   // UNICODE_TO_GBK[32326] := 16#8A56;
   // UNICODE_TO_GBK[32327] := 16#D476;
   // UNICODE_TO_GBK[32328] := 16#8A57;
   // UNICODE_TO_GBK[32329] := 16#D477;
   // UNICODE_TO_GBK[32330] := 16#8A58;
   // UNICODE_TO_GBK[32331] := 16#D478;
   // UNICODE_TO_GBK[32332] := 16#8A59;
   // UNICODE_TO_GBK[32333] := 16#D479;
   // UNICODE_TO_GBK[32334] := 16#8A5A;
   // UNICODE_TO_GBK[32335] := 16#D47A;
   // UNICODE_TO_GBK[32336] := 16#8A5B;
   // UNICODE_TO_GBK[32337] := 16#D47B;
   // UNICODE_TO_GBK[32338] := 16#8A5C;
   // UNICODE_TO_GBK[32339] := 16#D47C;
   // UNICODE_TO_GBK[32340] := 16#8A5D;
   // UNICODE_TO_GBK[32341] := 16#D47D;
   // UNICODE_TO_GBK[32342] := 16#8A5E;
   // UNICODE_TO_GBK[32343] := 16#D47E;
   // UNICODE_TO_GBK[32344] := 16#8A5F;
   // UNICODE_TO_GBK[32345] := 16#D480;
   // UNICODE_TO_GBK[32346] := 16#8A60;
   // UNICODE_TO_GBK[32347] := 16#D481;
   // UNICODE_TO_GBK[32348] := 16#8A61;
   // UNICODE_TO_GBK[32349] := 16#D482;
   // UNICODE_TO_GBK[32350] := 16#8A62;
   // UNICODE_TO_GBK[32351] := 16#D483;
   // UNICODE_TO_GBK[32352] := 16#8A63;
   // UNICODE_TO_GBK[32353] := 16#D484;
   // UNICODE_TO_GBK[32354] := 16#8A64;
   // UNICODE_TO_GBK[32355] := 16#D485;
   // UNICODE_TO_GBK[32356] := 16#8A65;
   // UNICODE_TO_GBK[32357] := 16#D486;
   // UNICODE_TO_GBK[32358] := 16#8A66;
   // UNICODE_TO_GBK[32359] := 16#D487;
   // UNICODE_TO_GBK[32360] := 16#8A67;
   // UNICODE_TO_GBK[32361] := 16#D488;
   // UNICODE_TO_GBK[32362] := 16#8A68;
   // UNICODE_TO_GBK[32363] := 16#D489;
   // UNICODE_TO_GBK[32364] := 16#8A69;
   // UNICODE_TO_GBK[32365] := 16#D48A;
   // UNICODE_TO_GBK[32366] := 16#8A6A;
   // UNICODE_TO_GBK[32367] := 16#D48B;
   // UNICODE_TO_GBK[32368] := 16#8A6B;
   // UNICODE_TO_GBK[32369] := 16#D48C;
   // UNICODE_TO_GBK[32370] := 16#8A6C;
   // UNICODE_TO_GBK[32371] := 16#D48D;
   // UNICODE_TO_GBK[32372] := 16#8A6D;
   // UNICODE_TO_GBK[32373] := 16#D48E;
   // UNICODE_TO_GBK[32374] := 16#8A6E;
   // UNICODE_TO_GBK[32375] := 16#D48F;
   // UNICODE_TO_GBK[32376] := 16#8A6F;
   // UNICODE_TO_GBK[32377] := 16#D490;
   // UNICODE_TO_GBK[32378] := 16#8A70;
   // UNICODE_TO_GBK[32379] := 16#D491;
   // UNICODE_TO_GBK[32380] := 16#8A71;
   // UNICODE_TO_GBK[32381] := 16#D492;
   // UNICODE_TO_GBK[32382] := 16#8A72;
   // UNICODE_TO_GBK[32383] := 16#D493;
   // UNICODE_TO_GBK[32384] := 16#8A73;
   // UNICODE_TO_GBK[32385] := 16#D494;
   // UNICODE_TO_GBK[32386] := 16#8A74;
   // UNICODE_TO_GBK[32387] := 16#D495;
   // UNICODE_TO_GBK[32388] := 16#8A75;
   // UNICODE_TO_GBK[32389] := 16#D496;
   // UNICODE_TO_GBK[32390] := 16#8A76;
   // UNICODE_TO_GBK[32391] := 16#D497;
   // UNICODE_TO_GBK[32392] := 16#8A77;
   // UNICODE_TO_GBK[32393] := 16#D498;
   // UNICODE_TO_GBK[32394] := 16#8A78;
   // UNICODE_TO_GBK[32395] := 16#D499;
   // UNICODE_TO_GBK[32396] := 16#8A79;
   // UNICODE_TO_GBK[32397] := 16#D5B2;
   // UNICODE_TO_GBK[32398] := 16#8A7A;
   // UNICODE_TO_GBK[32399] := 16#D49A;
   // UNICODE_TO_GBK[32400] := 16#8A7B;
   // UNICODE_TO_GBK[32401] := 16#D49B;
   // UNICODE_TO_GBK[32402] := 16#8A7C;
   // UNICODE_TO_GBK[32403] := 16#D49C;
   // UNICODE_TO_GBK[32404] := 16#8A7D;
   // UNICODE_TO_GBK[32405] := 16#D49D;
   // UNICODE_TO_GBK[32406] := 16#8A7E;
   // UNICODE_TO_GBK[32407] := 16#D49E;
   // UNICODE_TO_GBK[32408] := 16#8A7F;
   // UNICODE_TO_GBK[32409] := 16#D49F;
   // UNICODE_TO_GBK[32410] := 16#8A80;
   // UNICODE_TO_GBK[32411] := 16#D4A0;
   // UNICODE_TO_GBK[32412] := 16#8A81;
   // UNICODE_TO_GBK[32413] := 16#D540;
   // UNICODE_TO_GBK[32414] := 16#8A82;
   // UNICODE_TO_GBK[32415] := 16#D541;
   // UNICODE_TO_GBK[32416] := 16#8A83;
   // UNICODE_TO_GBK[32417] := 16#D542;
   // UNICODE_TO_GBK[32418] := 16#8A84;
   // UNICODE_TO_GBK[32419] := 16#D543;
   // UNICODE_TO_GBK[32420] := 16#8A85;
   // UNICODE_TO_GBK[32421] := 16#D544;
   // UNICODE_TO_GBK[32422] := 16#8A86;
   // UNICODE_TO_GBK[32423] := 16#D545;
   // UNICODE_TO_GBK[32424] := 16#8A87;
   // UNICODE_TO_GBK[32425] := 16#D546;
   // UNICODE_TO_GBK[32426] := 16#8A88;
   // UNICODE_TO_GBK[32427] := 16#D547;
   // UNICODE_TO_GBK[32428] := 16#8A89;
   // UNICODE_TO_GBK[32429] := 16#D3FE;
   // UNICODE_TO_GBK[32430] := 16#8A8A;
   // UNICODE_TO_GBK[32431] := 16#CCDC;
   // UNICODE_TO_GBK[32432] := 16#8A8B;
   // UNICODE_TO_GBK[32433] := 16#D548;
   // UNICODE_TO_GBK[32434] := 16#8A8C;
   // UNICODE_TO_GBK[32435] := 16#D549;
   // UNICODE_TO_GBK[32436] := 16#8A8D;
   // UNICODE_TO_GBK[32437] := 16#D54A;
   // UNICODE_TO_GBK[32438] := 16#8A8E;
   // UNICODE_TO_GBK[32439] := 16#D54B;
   // UNICODE_TO_GBK[32440] := 16#8A8F;
   // UNICODE_TO_GBK[32441] := 16#D54C;
   // UNICODE_TO_GBK[32442] := 16#8A90;
   // UNICODE_TO_GBK[32443] := 16#D54D;
   // UNICODE_TO_GBK[32444] := 16#8A91;
   // UNICODE_TO_GBK[32445] := 16#D54E;
   // UNICODE_TO_GBK[32446] := 16#8A92;
   // UNICODE_TO_GBK[32447] := 16#D54F;
   // UNICODE_TO_GBK[32448] := 16#8A93;
   // UNICODE_TO_GBK[32449] := 16#CAC4;
   // UNICODE_TO_GBK[32450] := 16#8A94;
   // UNICODE_TO_GBK[32451] := 16#D550;
   // UNICODE_TO_GBK[32452] := 16#8A95;
   // UNICODE_TO_GBK[32453] := 16#D551;
   // UNICODE_TO_GBK[32454] := 16#8A96;
   // UNICODE_TO_GBK[32455] := 16#D552;
   // UNICODE_TO_GBK[32456] := 16#8A97;
   // UNICODE_TO_GBK[32457] := 16#D553;
   // UNICODE_TO_GBK[32458] := 16#8A98;
   // UNICODE_TO_GBK[32459] := 16#D554;
   // UNICODE_TO_GBK[32460] := 16#8A99;
   // UNICODE_TO_GBK[32461] := 16#D555;
   // UNICODE_TO_GBK[32462] := 16#8A9A;
   // UNICODE_TO_GBK[32463] := 16#D556;
   // UNICODE_TO_GBK[32464] := 16#8A9B;
   // UNICODE_TO_GBK[32465] := 16#D557;
   // UNICODE_TO_GBK[32466] := 16#8A9C;
   // UNICODE_TO_GBK[32467] := 16#D558;
   // UNICODE_TO_GBK[32468] := 16#8A9D;
   // UNICODE_TO_GBK[32469] := 16#D559;
   // UNICODE_TO_GBK[32470] := 16#8A9E;
   // UNICODE_TO_GBK[32471] := 16#D55A;
   // UNICODE_TO_GBK[32472] := 16#8A9F;
   // UNICODE_TO_GBK[32473] := 16#D55B;
   // UNICODE_TO_GBK[32474] := 16#8AA0;
   // UNICODE_TO_GBK[32475] := 16#D55C;
   // UNICODE_TO_GBK[32476] := 16#8AA1;
   // UNICODE_TO_GBK[32477] := 16#D55D;
   // UNICODE_TO_GBK[32478] := 16#8AA2;
   // UNICODE_TO_GBK[32479] := 16#D55E;
   // UNICODE_TO_GBK[32480] := 16#8AA3;
   // UNICODE_TO_GBK[32481] := 16#D55F;
   // UNICODE_TO_GBK[32482] := 16#8AA4;
   // UNICODE_TO_GBK[32483] := 16#D560;
   // UNICODE_TO_GBK[32484] := 16#8AA5;
   // UNICODE_TO_GBK[32485] := 16#D561;
   // UNICODE_TO_GBK[32486] := 16#8AA6;
   // UNICODE_TO_GBK[32487] := 16#D562;
   // UNICODE_TO_GBK[32488] := 16#8AA7;
   // UNICODE_TO_GBK[32489] := 16#D563;
   // UNICODE_TO_GBK[32490] := 16#8AA8;
   // UNICODE_TO_GBK[32491] := 16#D564;
   // UNICODE_TO_GBK[32492] := 16#8AA9;
   // UNICODE_TO_GBK[32493] := 16#D565;
   // UNICODE_TO_GBK[32494] := 16#8AAA;
   // UNICODE_TO_GBK[32495] := 16#D566;
   // UNICODE_TO_GBK[32496] := 16#8AAB;
   // UNICODE_TO_GBK[32497] := 16#D567;
   // UNICODE_TO_GBK[32498] := 16#8AAC;
   // UNICODE_TO_GBK[32499] := 16#D568;
   // UNICODE_TO_GBK[32500] := 16#8AAD;
   // UNICODE_TO_GBK[32501] := 16#D569;
   // UNICODE_TO_GBK[32502] := 16#8AAE;
   // UNICODE_TO_GBK[32503] := 16#D56A;
   // UNICODE_TO_GBK[32504] := 16#8AAF;
   // UNICODE_TO_GBK[32505] := 16#D56B;
   // UNICODE_TO_GBK[32506] := 16#8AB0;
   // UNICODE_TO_GBK[32507] := 16#D56C;
   // UNICODE_TO_GBK[32508] := 16#8AB1;
   // UNICODE_TO_GBK[32509] := 16#D56D;
   // UNICODE_TO_GBK[32510] := 16#8AB2;
   // UNICODE_TO_GBK[32511] := 16#D56E;
   // UNICODE_TO_GBK[32512] := 16#8AB3;
   // UNICODE_TO_GBK[32513] := 16#D56F;
   // UNICODE_TO_GBK[32514] := 16#8AB4;
   // UNICODE_TO_GBK[32515] := 16#D570;
   // UNICODE_TO_GBK[32516] := 16#8AB5;
   // UNICODE_TO_GBK[32517] := 16#D571;
   // UNICODE_TO_GBK[32518] := 16#8AB6;
   // UNICODE_TO_GBK[32519] := 16#D572;
   // UNICODE_TO_GBK[32520] := 16#8AB7;
   // UNICODE_TO_GBK[32521] := 16#D573;
   // UNICODE_TO_GBK[32522] := 16#8AB8;
   // UNICODE_TO_GBK[32523] := 16#D574;
   // UNICODE_TO_GBK[32524] := 16#8AB9;
   // UNICODE_TO_GBK[32525] := 16#D575;
   // UNICODE_TO_GBK[32526] := 16#8ABA;
   // UNICODE_TO_GBK[32527] := 16#D576;
   // UNICODE_TO_GBK[32528] := 16#8ABB;
   // UNICODE_TO_GBK[32529] := 16#D577;
   // UNICODE_TO_GBK[32530] := 16#8ABC;
   // UNICODE_TO_GBK[32531] := 16#D578;
   // UNICODE_TO_GBK[32532] := 16#8ABD;
   // UNICODE_TO_GBK[32533] := 16#D579;
   // UNICODE_TO_GBK[32534] := 16#8ABE;
   // UNICODE_TO_GBK[32535] := 16#D57A;
   // UNICODE_TO_GBK[32536] := 16#8ABF;
   // UNICODE_TO_GBK[32537] := 16#D57B;
   // UNICODE_TO_GBK[32538] := 16#8AC0;
   // UNICODE_TO_GBK[32539] := 16#D57C;
   // UNICODE_TO_GBK[32540] := 16#8AC1;
   // UNICODE_TO_GBK[32541] := 16#D57D;
   // UNICODE_TO_GBK[32542] := 16#8AC2;
   // UNICODE_TO_GBK[32543] := 16#D57E;
   // UNICODE_TO_GBK[32544] := 16#8AC3;
   // UNICODE_TO_GBK[32545] := 16#D580;
   // UNICODE_TO_GBK[32546] := 16#8AC4;
   // UNICODE_TO_GBK[32547] := 16#D581;
   // UNICODE_TO_GBK[32548] := 16#8AC5;
   // UNICODE_TO_GBK[32549] := 16#D582;
   // UNICODE_TO_GBK[32550] := 16#8AC6;
   // UNICODE_TO_GBK[32551] := 16#D583;
   // UNICODE_TO_GBK[32552] := 16#8AC7;
   // UNICODE_TO_GBK[32553] := 16#D584;
   // UNICODE_TO_GBK[32554] := 16#8AC8;
   // UNICODE_TO_GBK[32555] := 16#D585;
   // UNICODE_TO_GBK[32556] := 16#8AC9;
   // UNICODE_TO_GBK[32557] := 16#D586;
   // UNICODE_TO_GBK[32558] := 16#8ACA;
   // UNICODE_TO_GBK[32559] := 16#D587;
   // UNICODE_TO_GBK[32560] := 16#8ACB;
   // UNICODE_TO_GBK[32561] := 16#D588;
   // UNICODE_TO_GBK[32562] := 16#8ACC;
   // UNICODE_TO_GBK[32563] := 16#D589;
   // UNICODE_TO_GBK[32564] := 16#8ACD;
   // UNICODE_TO_GBK[32565] := 16#D58A;
   // UNICODE_TO_GBK[32566] := 16#8ACE;
   // UNICODE_TO_GBK[32567] := 16#D58B;
   // UNICODE_TO_GBK[32568] := 16#8ACF;
   // UNICODE_TO_GBK[32569] := 16#D58C;
   // UNICODE_TO_GBK[32570] := 16#8AD0;
   // UNICODE_TO_GBK[32571] := 16#D58D;
   // UNICODE_TO_GBK[32572] := 16#8AD1;
   // UNICODE_TO_GBK[32573] := 16#D58E;
   // UNICODE_TO_GBK[32574] := 16#8AD2;
   // UNICODE_TO_GBK[32575] := 16#D58F;
   // UNICODE_TO_GBK[32576] := 16#8AD3;
   // UNICODE_TO_GBK[32577] := 16#D590;
   // UNICODE_TO_GBK[32578] := 16#8AD4;
   // UNICODE_TO_GBK[32579] := 16#D591;
   // UNICODE_TO_GBK[32580] := 16#8AD5;
   // UNICODE_TO_GBK[32581] := 16#D592;
   // UNICODE_TO_GBK[32582] := 16#8AD6;
   // UNICODE_TO_GBK[32583] := 16#D593;
   // UNICODE_TO_GBK[32584] := 16#8AD7;
   // UNICODE_TO_GBK[32585] := 16#D594;
   // UNICODE_TO_GBK[32586] := 16#8AD8;
   // UNICODE_TO_GBK[32587] := 16#D595;
   // UNICODE_TO_GBK[32588] := 16#8AD9;
   // UNICODE_TO_GBK[32589] := 16#D596;
   // UNICODE_TO_GBK[32590] := 16#8ADA;
   // UNICODE_TO_GBK[32591] := 16#D597;
   // UNICODE_TO_GBK[32592] := 16#8ADB;
   // UNICODE_TO_GBK[32593] := 16#D598;
   // UNICODE_TO_GBK[32594] := 16#8ADC;
   // UNICODE_TO_GBK[32595] := 16#D599;
   // UNICODE_TO_GBK[32596] := 16#8ADD;
   // UNICODE_TO_GBK[32597] := 16#D59A;
   // UNICODE_TO_GBK[32598] := 16#8ADE;
   // UNICODE_TO_GBK[32599] := 16#D59B;
   // UNICODE_TO_GBK[32600] := 16#8ADF;
   // UNICODE_TO_GBK[32601] := 16#D59C;
   // UNICODE_TO_GBK[32602] := 16#8AE0;
   // UNICODE_TO_GBK[32603] := 16#D59D;
   // UNICODE_TO_GBK[32604] := 16#8AE1;
   // UNICODE_TO_GBK[32605] := 16#D59E;
   // UNICODE_TO_GBK[32606] := 16#8AE2;
   // UNICODE_TO_GBK[32607] := 16#D59F;
   // UNICODE_TO_GBK[32608] := 16#8AE3;
   // UNICODE_TO_GBK[32609] := 16#D5A0;
   // UNICODE_TO_GBK[32610] := 16#8AE4;
   // UNICODE_TO_GBK[32611] := 16#D640;
   // UNICODE_TO_GBK[32612] := 16#8AE5;
   // UNICODE_TO_GBK[32613] := 16#D641;
   // UNICODE_TO_GBK[32614] := 16#8AE6;
   // UNICODE_TO_GBK[32615] := 16#D642;
   // UNICODE_TO_GBK[32616] := 16#8AE7;
   // UNICODE_TO_GBK[32617] := 16#D643;
   // UNICODE_TO_GBK[32618] := 16#8AE8;
   // UNICODE_TO_GBK[32619] := 16#D644;
   // UNICODE_TO_GBK[32620] := 16#8AE9;
   // UNICODE_TO_GBK[32621] := 16#D645;
   // UNICODE_TO_GBK[32622] := 16#8AEA;
   // UNICODE_TO_GBK[32623] := 16#D646;
   // UNICODE_TO_GBK[32624] := 16#8AEB;
   // UNICODE_TO_GBK[32625] := 16#D647;
   // UNICODE_TO_GBK[32626] := 16#8AEC;
   // UNICODE_TO_GBK[32627] := 16#D648;
   // UNICODE_TO_GBK[32628] := 16#8AED;
   // UNICODE_TO_GBK[32629] := 16#D649;
   // UNICODE_TO_GBK[32630] := 16#8AEE;
   // UNICODE_TO_GBK[32631] := 16#D64A;
   // UNICODE_TO_GBK[32632] := 16#8AEF;
   // UNICODE_TO_GBK[32633] := 16#D64B;
   // UNICODE_TO_GBK[32634] := 16#8AF0;
   // UNICODE_TO_GBK[32635] := 16#D64C;
   // UNICODE_TO_GBK[32636] := 16#8AF1;
   // UNICODE_TO_GBK[32637] := 16#D64D;
   // UNICODE_TO_GBK[32638] := 16#8AF2;
   // UNICODE_TO_GBK[32639] := 16#D64E;
   // UNICODE_TO_GBK[32640] := 16#8AF3;
   // UNICODE_TO_GBK[32641] := 16#D64F;
   // UNICODE_TO_GBK[32642] := 16#8AF4;
   // UNICODE_TO_GBK[32643] := 16#D650;
   // UNICODE_TO_GBK[32644] := 16#8AF5;
   // UNICODE_TO_GBK[32645] := 16#D651;
   // UNICODE_TO_GBK[32646] := 16#8AF6;
   // UNICODE_TO_GBK[32647] := 16#D652;
   // UNICODE_TO_GBK[32648] := 16#8AF7;
   // UNICODE_TO_GBK[32649] := 16#D653;
   // UNICODE_TO_GBK[32650] := 16#8AF8;
   // UNICODE_TO_GBK[32651] := 16#D654;
   // UNICODE_TO_GBK[32652] := 16#8AF9;
   // UNICODE_TO_GBK[32653] := 16#D655;
   // UNICODE_TO_GBK[32654] := 16#8AFA;
   // UNICODE_TO_GBK[32655] := 16#D656;
   // UNICODE_TO_GBK[32656] := 16#8AFB;
   // UNICODE_TO_GBK[32657] := 16#D657;
   // UNICODE_TO_GBK[32658] := 16#8AFC;
   // UNICODE_TO_GBK[32659] := 16#D658;
   // UNICODE_TO_GBK[32660] := 16#8AFD;
   // UNICODE_TO_GBK[32661] := 16#D659;
   // UNICODE_TO_GBK[32662] := 16#8AFE;
   // UNICODE_TO_GBK[32663] := 16#D65A;
   // UNICODE_TO_GBK[32664] := 16#8AFF;
   // UNICODE_TO_GBK[32665] := 16#D65B;
   // UNICODE_TO_GBK[32666] := 16#8B00;
   // UNICODE_TO_GBK[32667] := 16#D65C;
   // UNICODE_TO_GBK[32668] := 16#8B01;
   // UNICODE_TO_GBK[32669] := 16#D65D;
   // UNICODE_TO_GBK[32670] := 16#8B02;
   // UNICODE_TO_GBK[32671] := 16#D65E;
   // UNICODE_TO_GBK[32672] := 16#8B03;
   // UNICODE_TO_GBK[32673] := 16#D65F;
   // UNICODE_TO_GBK[32674] := 16#8B04;
   // UNICODE_TO_GBK[32675] := 16#D660;
   // UNICODE_TO_GBK[32676] := 16#8B05;
   // UNICODE_TO_GBK[32677] := 16#D661;
   // UNICODE_TO_GBK[32678] := 16#8B06;
   // UNICODE_TO_GBK[32679] := 16#D662;
   // UNICODE_TO_GBK[32680] := 16#8B07;
   // UNICODE_TO_GBK[32681] := 16#E5C0;
   // UNICODE_TO_GBK[32682] := 16#8B08;
   // UNICODE_TO_GBK[32683] := 16#D663;
   // UNICODE_TO_GBK[32684] := 16#8B09;
   // UNICODE_TO_GBK[32685] := 16#D664;
   // UNICODE_TO_GBK[32686] := 16#8B0A;
   // UNICODE_TO_GBK[32687] := 16#D665;
   // UNICODE_TO_GBK[32688] := 16#8B0B;
   // UNICODE_TO_GBK[32689] := 16#D666;
   // UNICODE_TO_GBK[32690] := 16#8B0C;
   // UNICODE_TO_GBK[32691] := 16#D667;
   // UNICODE_TO_GBK[32692] := 16#8B0D;
   // UNICODE_TO_GBK[32693] := 16#D668;
   // UNICODE_TO_GBK[32694] := 16#8B0E;
   // UNICODE_TO_GBK[32695] := 16#D669;
   // UNICODE_TO_GBK[32696] := 16#8B0F;
   // UNICODE_TO_GBK[32697] := 16#D66A;
   // UNICODE_TO_GBK[32698] := 16#8B10;
   // UNICODE_TO_GBK[32699] := 16#D66B;
   // UNICODE_TO_GBK[32700] := 16#8B11;
   // UNICODE_TO_GBK[32701] := 16#D66C;
   // UNICODE_TO_GBK[32702] := 16#8B12;
   // UNICODE_TO_GBK[32703] := 16#D66D;
   // UNICODE_TO_GBK[32704] := 16#8B13;
   // UNICODE_TO_GBK[32705] := 16#D66E;
   // UNICODE_TO_GBK[32706] := 16#8B14;
   // UNICODE_TO_GBK[32707] := 16#D66F;
   // UNICODE_TO_GBK[32708] := 16#8B15;
   // UNICODE_TO_GBK[32709] := 16#D670;
   // UNICODE_TO_GBK[32710] := 16#8B16;
   // UNICODE_TO_GBK[32711] := 16#D671;
   // UNICODE_TO_GBK[32712] := 16#8B17;
   // UNICODE_TO_GBK[32713] := 16#D672;
   // UNICODE_TO_GBK[32714] := 16#8B18;
   // UNICODE_TO_GBK[32715] := 16#D673;
   // UNICODE_TO_GBK[32716] := 16#8B19;
   // UNICODE_TO_GBK[32717] := 16#D674;
   // UNICODE_TO_GBK[32718] := 16#8B1A;
   // UNICODE_TO_GBK[32719] := 16#D675;
   // UNICODE_TO_GBK[32720] := 16#8B1B;
   // UNICODE_TO_GBK[32721] := 16#D676;
   // UNICODE_TO_GBK[32722] := 16#8B1C;
   // UNICODE_TO_GBK[32723] := 16#D677;
   // UNICODE_TO_GBK[32724] := 16#8B1D;
   // UNICODE_TO_GBK[32725] := 16#D678;
   // UNICODE_TO_GBK[32726] := 16#8B1E;
   // UNICODE_TO_GBK[32727] := 16#D679;
   // UNICODE_TO_GBK[32728] := 16#8B1F;
   // UNICODE_TO_GBK[32729] := 16#D67A;
   // UNICODE_TO_GBK[32730] := 16#8B20;
   // UNICODE_TO_GBK[32731] := 16#D67B;
   // UNICODE_TO_GBK[32732] := 16#8B21;
   // UNICODE_TO_GBK[32733] := 16#D67C;
   // UNICODE_TO_GBK[32734] := 16#8B22;
   // UNICODE_TO_GBK[32735] := 16#D67D;
   // UNICODE_TO_GBK[32736] := 16#8B23;
   // UNICODE_TO_GBK[32737] := 16#D67E;
   // UNICODE_TO_GBK[32738] := 16#8B24;
   // UNICODE_TO_GBK[32739] := 16#D680;
   // UNICODE_TO_GBK[32740] := 16#8B25;
   // UNICODE_TO_GBK[32741] := 16#D681;
   // UNICODE_TO_GBK[32742] := 16#8B26;
   // UNICODE_TO_GBK[32743] := 16#F6A5;
   // UNICODE_TO_GBK[32744] := 16#8B27;
   // UNICODE_TO_GBK[32745] := 16#D682;
   // UNICODE_TO_GBK[32746] := 16#8B28;
   // UNICODE_TO_GBK[32747] := 16#D683;
   // UNICODE_TO_GBK[32748] := 16#8B29;
   // UNICODE_TO_GBK[32749] := 16#D684;
   // UNICODE_TO_GBK[32750] := 16#8B2A;
   // UNICODE_TO_GBK[32751] := 16#D685;
   // UNICODE_TO_GBK[32752] := 16#8B2B;
   // UNICODE_TO_GBK[32753] := 16#D686;
   // UNICODE_TO_GBK[32754] := 16#8B2C;
   // UNICODE_TO_GBK[32755] := 16#D687;
   // UNICODE_TO_GBK[32756] := 16#8B2D;
   // UNICODE_TO_GBK[32757] := 16#D688;
   // UNICODE_TO_GBK[32758] := 16#8B2E;
   // UNICODE_TO_GBK[32759] := 16#D689;
   // UNICODE_TO_GBK[32760] := 16#8B2F;
   // UNICODE_TO_GBK[32761] := 16#D68A;
   // UNICODE_TO_GBK[32762] := 16#8B30;
   // UNICODE_TO_GBK[32763] := 16#D68B;
   // UNICODE_TO_GBK[32764] := 16#8B31;
   // UNICODE_TO_GBK[32765] := 16#D68C;
   // UNICODE_TO_GBK[32766] := 16#8B32;
   // UNICODE_TO_GBK[32767] := 16#D68D;
   // UNICODE_TO_GBK[32768] := 16#8B33;
   // UNICODE_TO_GBK[32769] := 16#D68E;
   // UNICODE_TO_GBK[32770] := 16#8B34;
   // UNICODE_TO_GBK[32771] := 16#D68F;
   // UNICODE_TO_GBK[32772] := 16#8B35;
   // UNICODE_TO_GBK[32773] := 16#D690;
   // UNICODE_TO_GBK[32774] := 16#8B36;
   // UNICODE_TO_GBK[32775] := 16#D691;
   // UNICODE_TO_GBK[32776] := 16#8B37;
   // UNICODE_TO_GBK[32777] := 16#D692;
   // UNICODE_TO_GBK[32778] := 16#8B38;
   // UNICODE_TO_GBK[32779] := 16#D693;
   // UNICODE_TO_GBK[32780] := 16#8B39;
   // UNICODE_TO_GBK[32781] := 16#D694;
   // UNICODE_TO_GBK[32782] := 16#8B3A;
   // UNICODE_TO_GBK[32783] := 16#D695;
   // UNICODE_TO_GBK[32784] := 16#8B3B;
   // UNICODE_TO_GBK[32785] := 16#D696;
   // UNICODE_TO_GBK[32786] := 16#8B3C;
   // UNICODE_TO_GBK[32787] := 16#D697;
   // UNICODE_TO_GBK[32788] := 16#8B3D;
   // UNICODE_TO_GBK[32789] := 16#D698;
   // UNICODE_TO_GBK[32790] := 16#8B3E;
   // UNICODE_TO_GBK[32791] := 16#D699;
   // UNICODE_TO_GBK[32792] := 16#8B3F;
   // UNICODE_TO_GBK[32793] := 16#D69A;
   // UNICODE_TO_GBK[32794] := 16#8B40;
   // UNICODE_TO_GBK[32795] := 16#D69B;
   // UNICODE_TO_GBK[32796] := 16#8B41;
   // UNICODE_TO_GBK[32797] := 16#D69C;
   // UNICODE_TO_GBK[32798] := 16#8B42;
   // UNICODE_TO_GBK[32799] := 16#D69D;
   // UNICODE_TO_GBK[32800] := 16#8B43;
   // UNICODE_TO_GBK[32801] := 16#D69E;
   // UNICODE_TO_GBK[32802] := 16#8B44;
   // UNICODE_TO_GBK[32803] := 16#D69F;
   // UNICODE_TO_GBK[32804] := 16#8B45;
   // UNICODE_TO_GBK[32805] := 16#D6A0;
   // UNICODE_TO_GBK[32806] := 16#8B46;
   // UNICODE_TO_GBK[32807] := 16#D740;
   // UNICODE_TO_GBK[32808] := 16#8B47;
   // UNICODE_TO_GBK[32809] := 16#D741;
   // UNICODE_TO_GBK[32810] := 16#8B48;
   // UNICODE_TO_GBK[32811] := 16#D742;
   // UNICODE_TO_GBK[32812] := 16#8B49;
   // UNICODE_TO_GBK[32813] := 16#D743;
   // UNICODE_TO_GBK[32814] := 16#8B4A;
   // UNICODE_TO_GBK[32815] := 16#D744;
   // UNICODE_TO_GBK[32816] := 16#8B4B;
   // UNICODE_TO_GBK[32817] := 16#D745;
   // UNICODE_TO_GBK[32818] := 16#8B4C;
   // UNICODE_TO_GBK[32819] := 16#D746;
   // UNICODE_TO_GBK[32820] := 16#8B4D;
   // UNICODE_TO_GBK[32821] := 16#D747;
   // UNICODE_TO_GBK[32822] := 16#8B4E;
   // UNICODE_TO_GBK[32823] := 16#D748;
   // UNICODE_TO_GBK[32824] := 16#8B4F;
   // UNICODE_TO_GBK[32825] := 16#D749;
   // UNICODE_TO_GBK[32826] := 16#8B50;
   // UNICODE_TO_GBK[32827] := 16#D74A;
   // UNICODE_TO_GBK[32828] := 16#8B51;
   // UNICODE_TO_GBK[32829] := 16#D74B;
   // UNICODE_TO_GBK[32830] := 16#8B52;
   // UNICODE_TO_GBK[32831] := 16#D74C;
   // UNICODE_TO_GBK[32832] := 16#8B53;
   // UNICODE_TO_GBK[32833] := 16#D74D;
   // UNICODE_TO_GBK[32834] := 16#8B54;
   // UNICODE_TO_GBK[32835] := 16#D74E;
   // UNICODE_TO_GBK[32836] := 16#8B55;
   // UNICODE_TO_GBK[32837] := 16#D74F;
   // UNICODE_TO_GBK[32838] := 16#8B56;
   // UNICODE_TO_GBK[32839] := 16#D750;
   // UNICODE_TO_GBK[32840] := 16#8B57;
   // UNICODE_TO_GBK[32841] := 16#D751;
   // UNICODE_TO_GBK[32842] := 16#8B58;
   // UNICODE_TO_GBK[32843] := 16#D752;
   // UNICODE_TO_GBK[32844] := 16#8B59;
   // UNICODE_TO_GBK[32845] := 16#D753;
   // UNICODE_TO_GBK[32846] := 16#8B5A;
   // UNICODE_TO_GBK[32847] := 16#D754;
   // UNICODE_TO_GBK[32848] := 16#8B5B;
   // UNICODE_TO_GBK[32849] := 16#D755;
   // UNICODE_TO_GBK[32850] := 16#8B5C;
   // UNICODE_TO_GBK[32851] := 16#D756;
   // UNICODE_TO_GBK[32852] := 16#8B5D;
   // UNICODE_TO_GBK[32853] := 16#D757;
   // UNICODE_TO_GBK[32854] := 16#8B5E;
   // UNICODE_TO_GBK[32855] := 16#D758;
   // UNICODE_TO_GBK[32856] := 16#8B5F;
   // UNICODE_TO_GBK[32857] := 16#D759;
   // UNICODE_TO_GBK[32858] := 16#8B60;
   // UNICODE_TO_GBK[32859] := 16#D75A;
   // UNICODE_TO_GBK[32860] := 16#8B61;
   // UNICODE_TO_GBK[32861] := 16#D75B;
   // UNICODE_TO_GBK[32862] := 16#8B62;
   // UNICODE_TO_GBK[32863] := 16#D75C;
   // UNICODE_TO_GBK[32864] := 16#8B63;
   // UNICODE_TO_GBK[32865] := 16#D75D;
   // UNICODE_TO_GBK[32866] := 16#8B64;
   // UNICODE_TO_GBK[32867] := 16#D75E;
   // UNICODE_TO_GBK[32868] := 16#8B65;
   // UNICODE_TO_GBK[32869] := 16#D75F;
   // UNICODE_TO_GBK[32870] := 16#8B66;
   // UNICODE_TO_GBK[32871] := 16#BEAF;
   // UNICODE_TO_GBK[32872] := 16#8B67;
   // UNICODE_TO_GBK[32873] := 16#D760;
   // UNICODE_TO_GBK[32874] := 16#8B68;
   // UNICODE_TO_GBK[32875] := 16#D761;
   // UNICODE_TO_GBK[32876] := 16#8B69;
   // UNICODE_TO_GBK[32877] := 16#D762;
   // UNICODE_TO_GBK[32878] := 16#8B6A;
   // UNICODE_TO_GBK[32879] := 16#D763;
   // UNICODE_TO_GBK[32880] := 16#8B6B;
   // UNICODE_TO_GBK[32881] := 16#D764;
   // UNICODE_TO_GBK[32882] := 16#8B6C;
   // UNICODE_TO_GBK[32883] := 16#C6A9;
   // UNICODE_TO_GBK[32884] := 16#8B6D;
   // UNICODE_TO_GBK[32885] := 16#D765;
   // UNICODE_TO_GBK[32886] := 16#8B6E;
   // UNICODE_TO_GBK[32887] := 16#D766;
   // UNICODE_TO_GBK[32888] := 16#8B6F;
   // UNICODE_TO_GBK[32889] := 16#D767;
   // UNICODE_TO_GBK[32890] := 16#8B70;
   // UNICODE_TO_GBK[32891] := 16#D768;
   // UNICODE_TO_GBK[32892] := 16#8B71;
   // UNICODE_TO_GBK[32893] := 16#D769;
   // UNICODE_TO_GBK[32894] := 16#8B72;
   // UNICODE_TO_GBK[32895] := 16#D76A;
   // UNICODE_TO_GBK[32896] := 16#8B73;
   // UNICODE_TO_GBK[32897] := 16#D76B;
   // UNICODE_TO_GBK[32898] := 16#8B74;
   // UNICODE_TO_GBK[32899] := 16#D76C;
   // UNICODE_TO_GBK[32900] := 16#8B75;
   // UNICODE_TO_GBK[32901] := 16#D76D;
   // UNICODE_TO_GBK[32902] := 16#8B76;
   // UNICODE_TO_GBK[32903] := 16#D76E;
   // UNICODE_TO_GBK[32904] := 16#8B77;
   // UNICODE_TO_GBK[32905] := 16#D76F;
   // UNICODE_TO_GBK[32906] := 16#8B78;
   // UNICODE_TO_GBK[32907] := 16#D770;
   // UNICODE_TO_GBK[32908] := 16#8B79;
   // UNICODE_TO_GBK[32909] := 16#D771;
   // UNICODE_TO_GBK[32910] := 16#8B7A;
   // UNICODE_TO_GBK[32911] := 16#D772;
   // UNICODE_TO_GBK[32912] := 16#8B7B;
   // UNICODE_TO_GBK[32913] := 16#D773;
   // UNICODE_TO_GBK[32914] := 16#8B7C;
   // UNICODE_TO_GBK[32915] := 16#D774;
   // UNICODE_TO_GBK[32916] := 16#8B7D;
   // UNICODE_TO_GBK[32917] := 16#D775;
   // UNICODE_TO_GBK[32918] := 16#8B7E;
   // UNICODE_TO_GBK[32919] := 16#D776;
   // UNICODE_TO_GBK[32920] := 16#8B7F;
   // UNICODE_TO_GBK[32921] := 16#D777;
   // UNICODE_TO_GBK[32922] := 16#8B80;
   // UNICODE_TO_GBK[32923] := 16#D778;
   // UNICODE_TO_GBK[32924] := 16#8B81;
   // UNICODE_TO_GBK[32925] := 16#D779;
   // UNICODE_TO_GBK[32926] := 16#8B82;
   // UNICODE_TO_GBK[32927] := 16#D77A;
   // UNICODE_TO_GBK[32928] := 16#8B83;
   // UNICODE_TO_GBK[32929] := 16#D77B;
   // UNICODE_TO_GBK[32930] := 16#8B84;
   // UNICODE_TO_GBK[32931] := 16#D77C;
   // UNICODE_TO_GBK[32932] := 16#8B85;
   // UNICODE_TO_GBK[32933] := 16#D77D;
   // UNICODE_TO_GBK[32934] := 16#8B86;
   // UNICODE_TO_GBK[32935] := 16#D77E;
   // UNICODE_TO_GBK[32936] := 16#8B87;
   // UNICODE_TO_GBK[32937] := 16#D780;
   // UNICODE_TO_GBK[32938] := 16#8B88;
   // UNICODE_TO_GBK[32939] := 16#D781;
   // UNICODE_TO_GBK[32940] := 16#8B89;
   // UNICODE_TO_GBK[32941] := 16#D782;
   // UNICODE_TO_GBK[32942] := 16#8B8A;
   // UNICODE_TO_GBK[32943] := 16#D783;
   // UNICODE_TO_GBK[32944] := 16#8B8B;
   // UNICODE_TO_GBK[32945] := 16#D784;
   // UNICODE_TO_GBK[32946] := 16#8B8C;
   // UNICODE_TO_GBK[32947] := 16#D785;
   // UNICODE_TO_GBK[32948] := 16#8B8D;
   // UNICODE_TO_GBK[32949] := 16#D786;
   // UNICODE_TO_GBK[32950] := 16#8B8E;
   // UNICODE_TO_GBK[32951] := 16#D787;
   // UNICODE_TO_GBK[32952] := 16#8B8F;
   // UNICODE_TO_GBK[32953] := 16#D788;
   // UNICODE_TO_GBK[32954] := 16#8B90;
   // UNICODE_TO_GBK[32955] := 16#D789;
   // UNICODE_TO_GBK[32956] := 16#8B91;
   // UNICODE_TO_GBK[32957] := 16#D78A;
   // UNICODE_TO_GBK[32958] := 16#8B92;
   // UNICODE_TO_GBK[32959] := 16#D78B;
   // UNICODE_TO_GBK[32960] := 16#8B93;
   // UNICODE_TO_GBK[32961] := 16#D78C;
   // UNICODE_TO_GBK[32962] := 16#8B94;
   // UNICODE_TO_GBK[32963] := 16#D78D;
   // UNICODE_TO_GBK[32964] := 16#8B95;
   // UNICODE_TO_GBK[32965] := 16#D78E;
   // UNICODE_TO_GBK[32966] := 16#8B96;
   // UNICODE_TO_GBK[32967] := 16#D78F;
   // UNICODE_TO_GBK[32968] := 16#8B97;
   // UNICODE_TO_GBK[32969] := 16#D790;
   // UNICODE_TO_GBK[32970] := 16#8B98;
   // UNICODE_TO_GBK[32971] := 16#D791;
   // UNICODE_TO_GBK[32972] := 16#8B99;
   // UNICODE_TO_GBK[32973] := 16#D792;
   // UNICODE_TO_GBK[32974] := 16#8B9A;
   // UNICODE_TO_GBK[32975] := 16#D793;
   // UNICODE_TO_GBK[32976] := 16#8B9B;
   // UNICODE_TO_GBK[32977] := 16#D794;
   // UNICODE_TO_GBK[32978] := 16#8B9C;
   // UNICODE_TO_GBK[32979] := 16#D795;
   // UNICODE_TO_GBK[32980] := 16#8B9D;
   // UNICODE_TO_GBK[32981] := 16#D796;
   // UNICODE_TO_GBK[32982] := 16#8B9E;
   // UNICODE_TO_GBK[32983] := 16#D797;
   // UNICODE_TO_GBK[32984] := 16#8B9F;
   // UNICODE_TO_GBK[32985] := 16#D798;
   // UNICODE_TO_GBK[32986] := 16#8BA0;
   // UNICODE_TO_GBK[32987] := 16#DAA5;
   // UNICODE_TO_GBK[32988] := 16#8BA1;
   // UNICODE_TO_GBK[32989] := 16#BCC6;
   // UNICODE_TO_GBK[32990] := 16#8BA2;
   // UNICODE_TO_GBK[32991] := 16#B6A9;
   // UNICODE_TO_GBK[32992] := 16#8BA3;
   // UNICODE_TO_GBK[32993] := 16#B8BC;
   // UNICODE_TO_GBK[32994] := 16#8BA4;
   // UNICODE_TO_GBK[32995] := 16#C8CF;
   // UNICODE_TO_GBK[32996] := 16#8BA5;
   // UNICODE_TO_GBK[32997] := 16#BCA5;
   // UNICODE_TO_GBK[32998] := 16#8BA6;
   // UNICODE_TO_GBK[32999] := 16#DAA6;
   // UNICODE_TO_GBK[33000] := 16#8BA7;
   // UNICODE_TO_GBK[33001] := 16#DAA7;
   // UNICODE_TO_GBK[33002] := 16#8BA8;
   // UNICODE_TO_GBK[33003] := 16#CCD6;
   // UNICODE_TO_GBK[33004] := 16#8BA9;
   // UNICODE_TO_GBK[33005] := 16#C8C3;
   // UNICODE_TO_GBK[33006] := 16#8BAA;
   // UNICODE_TO_GBK[33007] := 16#DAA8;
   // UNICODE_TO_GBK[33008] := 16#8BAB;
   // UNICODE_TO_GBK[33009] := 16#C6FD;
   // UNICODE_TO_GBK[33010] := 16#8BAC;
   // UNICODE_TO_GBK[33011] := 16#D799;
   // UNICODE_TO_GBK[33012] := 16#8BAD;
   // UNICODE_TO_GBK[33013] := 16#D1B5;
   // UNICODE_TO_GBK[33014] := 16#8BAE;
   // UNICODE_TO_GBK[33015] := 16#D2E9;
   // UNICODE_TO_GBK[33016] := 16#8BAF;
   // UNICODE_TO_GBK[33017] := 16#D1B6;
   // UNICODE_TO_GBK[33018] := 16#8BB0;
   // UNICODE_TO_GBK[33019] := 16#BCC7;
   // UNICODE_TO_GBK[33020] := 16#8BB1;
   // UNICODE_TO_GBK[33021] := 16#D79A;
   // UNICODE_TO_GBK[33022] := 16#8BB2;
   // UNICODE_TO_GBK[33023] := 16#BDB2;
   // UNICODE_TO_GBK[33024] := 16#8BB3;
   // UNICODE_TO_GBK[33025] := 16#BBE4;
   // UNICODE_TO_GBK[33026] := 16#8BB4;
   // UNICODE_TO_GBK[33027] := 16#DAA9;
   // UNICODE_TO_GBK[33028] := 16#8BB5;
   // UNICODE_TO_GBK[33029] := 16#DAAA;
   // UNICODE_TO_GBK[33030] := 16#8BB6;
   // UNICODE_TO_GBK[33031] := 16#D1C8;
   // UNICODE_TO_GBK[33032] := 16#8BB7;
   // UNICODE_TO_GBK[33033] := 16#DAAB;
   // UNICODE_TO_GBK[33034] := 16#8BB8;
   // UNICODE_TO_GBK[33035] := 16#D0ED;
   // UNICODE_TO_GBK[33036] := 16#8BB9;
   // UNICODE_TO_GBK[33037] := 16#B6EF;
   // UNICODE_TO_GBK[33038] := 16#8BBA;
   // UNICODE_TO_GBK[33039] := 16#C2DB;
   // UNICODE_TO_GBK[33040] := 16#8BBB;
   // UNICODE_TO_GBK[33041] := 16#D79B;
   // UNICODE_TO_GBK[33042] := 16#8BBC;
   // UNICODE_TO_GBK[33043] := 16#CBCF;
   // UNICODE_TO_GBK[33044] := 16#8BBD;
   // UNICODE_TO_GBK[33045] := 16#B7ED;
   // UNICODE_TO_GBK[33046] := 16#8BBE;
   // UNICODE_TO_GBK[33047] := 16#C9E8;
   // UNICODE_TO_GBK[33048] := 16#8BBF;
   // UNICODE_TO_GBK[33049] := 16#B7C3;
   // UNICODE_TO_GBK[33050] := 16#8BC0;
   // UNICODE_TO_GBK[33051] := 16#BEF7;
   // UNICODE_TO_GBK[33052] := 16#8BC1;
   // UNICODE_TO_GBK[33053] := 16#D6A4;
   // UNICODE_TO_GBK[33054] := 16#8BC2;
   // UNICODE_TO_GBK[33055] := 16#DAAC;
   // UNICODE_TO_GBK[33056] := 16#8BC3;
   // UNICODE_TO_GBK[33057] := 16#DAAD;
   // UNICODE_TO_GBK[33058] := 16#8BC4;
   // UNICODE_TO_GBK[33059] := 16#C6C0;
   // UNICODE_TO_GBK[33060] := 16#8BC5;
   // UNICODE_TO_GBK[33061] := 16#D7E7;
   // UNICODE_TO_GBK[33062] := 16#8BC6;
   // UNICODE_TO_GBK[33063] := 16#CAB6;
   // UNICODE_TO_GBK[33064] := 16#8BC7;
   // UNICODE_TO_GBK[33065] := 16#D79C;
   // UNICODE_TO_GBK[33066] := 16#8BC8;
   // UNICODE_TO_GBK[33067] := 16#D5A9;
   // UNICODE_TO_GBK[33068] := 16#8BC9;
   // UNICODE_TO_GBK[33069] := 16#CBDF;
   // UNICODE_TO_GBK[33070] := 16#8BCA;
   // UNICODE_TO_GBK[33071] := 16#D5EF;
   // UNICODE_TO_GBK[33072] := 16#8BCB;
   // UNICODE_TO_GBK[33073] := 16#DAAE;
   // UNICODE_TO_GBK[33074] := 16#8BCC;
   // UNICODE_TO_GBK[33075] := 16#D6DF;
   // UNICODE_TO_GBK[33076] := 16#8BCD;
   // UNICODE_TO_GBK[33077] := 16#B4CA;
   // UNICODE_TO_GBK[33078] := 16#8BCE;
   // UNICODE_TO_GBK[33079] := 16#DAB0;
   // UNICODE_TO_GBK[33080] := 16#8BCF;
   // UNICODE_TO_GBK[33081] := 16#DAAF;
   // UNICODE_TO_GBK[33082] := 16#8BD0;
   // UNICODE_TO_GBK[33083] := 16#D79D;
   // UNICODE_TO_GBK[33084] := 16#8BD1;
   // UNICODE_TO_GBK[33085] := 16#D2EB;
   // UNICODE_TO_GBK[33086] := 16#8BD2;
   // UNICODE_TO_GBK[33087] := 16#DAB1;
   // UNICODE_TO_GBK[33088] := 16#8BD3;
   // UNICODE_TO_GBK[33089] := 16#DAB2;
   // UNICODE_TO_GBK[33090] := 16#8BD4;
   // UNICODE_TO_GBK[33091] := 16#DAB3;
   // UNICODE_TO_GBK[33092] := 16#8BD5;
   // UNICODE_TO_GBK[33093] := 16#CAD4;
   // UNICODE_TO_GBK[33094] := 16#8BD6;
   // UNICODE_TO_GBK[33095] := 16#DAB4;
   // UNICODE_TO_GBK[33096] := 16#8BD7;
   // UNICODE_TO_GBK[33097] := 16#CAAB;
   // UNICODE_TO_GBK[33098] := 16#8BD8;
   // UNICODE_TO_GBK[33099] := 16#DAB5;
   // UNICODE_TO_GBK[33100] := 16#8BD9;
   // UNICODE_TO_GBK[33101] := 16#DAB6;
   // UNICODE_TO_GBK[33102] := 16#8BDA;
   // UNICODE_TO_GBK[33103] := 16#B3CF;
   // UNICODE_TO_GBK[33104] := 16#8BDB;
   // UNICODE_TO_GBK[33105] := 16#D6EF;
   // UNICODE_TO_GBK[33106] := 16#8BDC;
   // UNICODE_TO_GBK[33107] := 16#DAB7;
   // UNICODE_TO_GBK[33108] := 16#8BDD;
   // UNICODE_TO_GBK[33109] := 16#BBB0;
   // UNICODE_TO_GBK[33110] := 16#8BDE;
   // UNICODE_TO_GBK[33111] := 16#B5AE;
   // UNICODE_TO_GBK[33112] := 16#8BDF;
   // UNICODE_TO_GBK[33113] := 16#DAB8;
   // UNICODE_TO_GBK[33114] := 16#8BE0;
   // UNICODE_TO_GBK[33115] := 16#DAB9;
   // UNICODE_TO_GBK[33116] := 16#8BE1;
   // UNICODE_TO_GBK[33117] := 16#B9EE;
   // UNICODE_TO_GBK[33118] := 16#8BE2;
   // UNICODE_TO_GBK[33119] := 16#D1AF;
   // UNICODE_TO_GBK[33120] := 16#8BE3;
   // UNICODE_TO_GBK[33121] := 16#D2E8;
   // UNICODE_TO_GBK[33122] := 16#8BE4;
   // UNICODE_TO_GBK[33123] := 16#DABA;
   // UNICODE_TO_GBK[33124] := 16#8BE5;
   // UNICODE_TO_GBK[33125] := 16#B8C3;
   // UNICODE_TO_GBK[33126] := 16#8BE6;
   // UNICODE_TO_GBK[33127] := 16#CFEA;
   // UNICODE_TO_GBK[33128] := 16#8BE7;
   // UNICODE_TO_GBK[33129] := 16#B2EF;
   // UNICODE_TO_GBK[33130] := 16#8BE8;
   // UNICODE_TO_GBK[33131] := 16#DABB;
   // UNICODE_TO_GBK[33132] := 16#8BE9;
   // UNICODE_TO_GBK[33133] := 16#DABC;
   // UNICODE_TO_GBK[33134] := 16#8BEA;
   // UNICODE_TO_GBK[33135] := 16#D79E;
   // UNICODE_TO_GBK[33136] := 16#8BEB;
   // UNICODE_TO_GBK[33137] := 16#BDEB;
   // UNICODE_TO_GBK[33138] := 16#8BEC;
   // UNICODE_TO_GBK[33139] := 16#CEDC;
   // UNICODE_TO_GBK[33140] := 16#8BED;
   // UNICODE_TO_GBK[33141] := 16#D3EF;
   // UNICODE_TO_GBK[33142] := 16#8BEE;
   // UNICODE_TO_GBK[33143] := 16#DABD;
   // UNICODE_TO_GBK[33144] := 16#8BEF;
   // UNICODE_TO_GBK[33145] := 16#CEF3;
   // UNICODE_TO_GBK[33146] := 16#8BF0;
   // UNICODE_TO_GBK[33147] := 16#DABE;
   // UNICODE_TO_GBK[33148] := 16#8BF1;
   // UNICODE_TO_GBK[33149] := 16#D3D5;
   // UNICODE_TO_GBK[33150] := 16#8BF2;
   // UNICODE_TO_GBK[33151] := 16#BBE5;
   // UNICODE_TO_GBK[33152] := 16#8BF3;
   // UNICODE_TO_GBK[33153] := 16#DABF;
   // UNICODE_TO_GBK[33154] := 16#8BF4;
   // UNICODE_TO_GBK[33155] := 16#CBB5;
   // UNICODE_TO_GBK[33156] := 16#8BF5;
   // UNICODE_TO_GBK[33157] := 16#CBD0;
   // UNICODE_TO_GBK[33158] := 16#8BF6;
   // UNICODE_TO_GBK[33159] := 16#DAC0;
   // UNICODE_TO_GBK[33160] := 16#8BF7;
   // UNICODE_TO_GBK[33161] := 16#C7EB;
   // UNICODE_TO_GBK[33162] := 16#8BF8;
   // UNICODE_TO_GBK[33163] := 16#D6EE;
   // UNICODE_TO_GBK[33164] := 16#8BF9;
   // UNICODE_TO_GBK[33165] := 16#DAC1;
   // UNICODE_TO_GBK[33166] := 16#8BFA;
   // UNICODE_TO_GBK[33167] := 16#C5B5;
   // UNICODE_TO_GBK[33168] := 16#8BFB;
   // UNICODE_TO_GBK[33169] := 16#B6C1;
   // UNICODE_TO_GBK[33170] := 16#8BFC;
   // UNICODE_TO_GBK[33171] := 16#DAC2;
   // UNICODE_TO_GBK[33172] := 16#8BFD;
   // UNICODE_TO_GBK[33173] := 16#B7CC;
   // UNICODE_TO_GBK[33174] := 16#8BFE;
   // UNICODE_TO_GBK[33175] := 16#BFCE;
   // UNICODE_TO_GBK[33176] := 16#8BFF;
   // UNICODE_TO_GBK[33177] := 16#DAC3;
   // UNICODE_TO_GBK[33178] := 16#8C00;
   // UNICODE_TO_GBK[33179] := 16#DAC4;
   // UNICODE_TO_GBK[33180] := 16#8C01;
   // UNICODE_TO_GBK[33181] := 16#CBAD;
   // UNICODE_TO_GBK[33182] := 16#8C02;
   // UNICODE_TO_GBK[33183] := 16#DAC5;
   // UNICODE_TO_GBK[33184] := 16#8C03;
   // UNICODE_TO_GBK[33185] := 16#B5F7;
   // UNICODE_TO_GBK[33186] := 16#8C04;
   // UNICODE_TO_GBK[33187] := 16#DAC6;
   // UNICODE_TO_GBK[33188] := 16#8C05;
   // UNICODE_TO_GBK[33189] := 16#C1C2;
   // UNICODE_TO_GBK[33190] := 16#8C06;
   // UNICODE_TO_GBK[33191] := 16#D7BB;
   // UNICODE_TO_GBK[33192] := 16#8C07;
   // UNICODE_TO_GBK[33193] := 16#DAC7;
   // UNICODE_TO_GBK[33194] := 16#8C08;
   // UNICODE_TO_GBK[33195] := 16#CCB8;
   // UNICODE_TO_GBK[33196] := 16#8C09;
   // UNICODE_TO_GBK[33197] := 16#D79F;
   // UNICODE_TO_GBK[33198] := 16#8C0A;
   // UNICODE_TO_GBK[33199] := 16#D2EA;
   // UNICODE_TO_GBK[33200] := 16#8C0B;
   // UNICODE_TO_GBK[33201] := 16#C4B1;
   // UNICODE_TO_GBK[33202] := 16#8C0C;
   // UNICODE_TO_GBK[33203] := 16#DAC8;
   // UNICODE_TO_GBK[33204] := 16#8C0D;
   // UNICODE_TO_GBK[33205] := 16#B5FD;
   // UNICODE_TO_GBK[33206] := 16#8C0E;
   // UNICODE_TO_GBK[33207] := 16#BBD1;
   // UNICODE_TO_GBK[33208] := 16#8C0F;
   // UNICODE_TO_GBK[33209] := 16#DAC9;
   // UNICODE_TO_GBK[33210] := 16#8C10;
   // UNICODE_TO_GBK[33211] := 16#D0B3;
   // UNICODE_TO_GBK[33212] := 16#8C11;
   // UNICODE_TO_GBK[33213] := 16#DACA;
   // UNICODE_TO_GBK[33214] := 16#8C12;
   // UNICODE_TO_GBK[33215] := 16#DACB;
   // UNICODE_TO_GBK[33216] := 16#8C13;
   // UNICODE_TO_GBK[33217] := 16#CEBD;
   // UNICODE_TO_GBK[33218] := 16#8C14;
   // UNICODE_TO_GBK[33219] := 16#DACC;
   // UNICODE_TO_GBK[33220] := 16#8C15;
   // UNICODE_TO_GBK[33221] := 16#DACD;
   // UNICODE_TO_GBK[33222] := 16#8C16;
   // UNICODE_TO_GBK[33223] := 16#DACE;
   // UNICODE_TO_GBK[33224] := 16#8C17;
   // UNICODE_TO_GBK[33225] := 16#B2F7;
   // UNICODE_TO_GBK[33226] := 16#8C18;
   // UNICODE_TO_GBK[33227] := 16#DAD1;
   // UNICODE_TO_GBK[33228] := 16#8C19;
   // UNICODE_TO_GBK[33229] := 16#DACF;
   // UNICODE_TO_GBK[33230] := 16#8C1A;
   // UNICODE_TO_GBK[33231] := 16#D1E8;
   // UNICODE_TO_GBK[33232] := 16#8C1B;
   // UNICODE_TO_GBK[33233] := 16#DAD0;
   // UNICODE_TO_GBK[33234] := 16#8C1C;
   // UNICODE_TO_GBK[33235] := 16#C3D5;
   // UNICODE_TO_GBK[33236] := 16#8C1D;
   // UNICODE_TO_GBK[33237] := 16#DAD2;
   // UNICODE_TO_GBK[33238] := 16#8C1E;
   // UNICODE_TO_GBK[33239] := 16#D7A0;
   // UNICODE_TO_GBK[33240] := 16#8C1F;
   // UNICODE_TO_GBK[33241] := 16#DAD3;
   // UNICODE_TO_GBK[33242] := 16#8C20;
   // UNICODE_TO_GBK[33243] := 16#DAD4;
   // UNICODE_TO_GBK[33244] := 16#8C21;
   // UNICODE_TO_GBK[33245] := 16#DAD5;
   // UNICODE_TO_GBK[33246] := 16#8C22;
   // UNICODE_TO_GBK[33247] := 16#D0BB;
   // UNICODE_TO_GBK[33248] := 16#8C23;
   // UNICODE_TO_GBK[33249] := 16#D2A5;
   // UNICODE_TO_GBK[33250] := 16#8C24;
   // UNICODE_TO_GBK[33251] := 16#B0F9;
   // UNICODE_TO_GBK[33252] := 16#8C25;
   // UNICODE_TO_GBK[33253] := 16#DAD6;
   // UNICODE_TO_GBK[33254] := 16#8C26;
   // UNICODE_TO_GBK[33255] := 16#C7AB;
   // UNICODE_TO_GBK[33256] := 16#8C27;
   // UNICODE_TO_GBK[33257] := 16#DAD7;
   // UNICODE_TO_GBK[33258] := 16#8C28;
   // UNICODE_TO_GBK[33259] := 16#BDF7;
   // UNICODE_TO_GBK[33260] := 16#8C29;
   // UNICODE_TO_GBK[33261] := 16#C3A1;
   // UNICODE_TO_GBK[33262] := 16#8C2A;
   // UNICODE_TO_GBK[33263] := 16#DAD8;
   // UNICODE_TO_GBK[33264] := 16#8C2B;
   // UNICODE_TO_GBK[33265] := 16#DAD9;
   // UNICODE_TO_GBK[33266] := 16#8C2C;
   // UNICODE_TO_GBK[33267] := 16#C3FD;
   // UNICODE_TO_GBK[33268] := 16#8C2D;
   // UNICODE_TO_GBK[33269] := 16#CCB7;
   // UNICODE_TO_GBK[33270] := 16#8C2E;
   // UNICODE_TO_GBK[33271] := 16#DADA;
   // UNICODE_TO_GBK[33272] := 16#8C2F;
   // UNICODE_TO_GBK[33273] := 16#DADB;
   // UNICODE_TO_GBK[33274] := 16#8C30;
   // UNICODE_TO_GBK[33275] := 16#C0BE;
   // UNICODE_TO_GBK[33276] := 16#8C31;
   // UNICODE_TO_GBK[33277] := 16#C6D7;
   // UNICODE_TO_GBK[33278] := 16#8C32;
   // UNICODE_TO_GBK[33279] := 16#DADC;
   // UNICODE_TO_GBK[33280] := 16#8C33;
   // UNICODE_TO_GBK[33281] := 16#DADD;
   // UNICODE_TO_GBK[33282] := 16#8C34;
   // UNICODE_TO_GBK[33283] := 16#C7B4;
   // UNICODE_TO_GBK[33284] := 16#8C35;
   // UNICODE_TO_GBK[33285] := 16#DADE;
   // UNICODE_TO_GBK[33286] := 16#8C36;
   // UNICODE_TO_GBK[33287] := 16#DADF;
   // UNICODE_TO_GBK[33288] := 16#8C37;
   // UNICODE_TO_GBK[33289] := 16#B9C8;
   // UNICODE_TO_GBK[33290] := 16#8C38;
   // UNICODE_TO_GBK[33291] := 16#D840;
   // UNICODE_TO_GBK[33292] := 16#8C39;
   // UNICODE_TO_GBK[33293] := 16#D841;
   // UNICODE_TO_GBK[33294] := 16#8C3A;
   // UNICODE_TO_GBK[33295] := 16#D842;
   // UNICODE_TO_GBK[33296] := 16#8C3B;
   // UNICODE_TO_GBK[33297] := 16#D843;
   // UNICODE_TO_GBK[33298] := 16#8C3C;
   // UNICODE_TO_GBK[33299] := 16#D844;
   // UNICODE_TO_GBK[33300] := 16#8C3D;
   // UNICODE_TO_GBK[33301] := 16#D845;
   // UNICODE_TO_GBK[33302] := 16#8C3E;
   // UNICODE_TO_GBK[33303] := 16#D846;
   // UNICODE_TO_GBK[33304] := 16#8C3F;
   // UNICODE_TO_GBK[33305] := 16#D847;
   // UNICODE_TO_GBK[33306] := 16#8C40;
   // UNICODE_TO_GBK[33307] := 16#D848;
   // UNICODE_TO_GBK[33308] := 16#8C41;
   // UNICODE_TO_GBK[33309] := 16#BBED;
   // UNICODE_TO_GBK[33310] := 16#8C42;
   // UNICODE_TO_GBK[33311] := 16#D849;
   // UNICODE_TO_GBK[33312] := 16#8C43;
   // UNICODE_TO_GBK[33313] := 16#D84A;
   // UNICODE_TO_GBK[33314] := 16#8C44;
   // UNICODE_TO_GBK[33315] := 16#D84B;
   // UNICODE_TO_GBK[33316] := 16#8C45;
   // UNICODE_TO_GBK[33317] := 16#D84C;
   // UNICODE_TO_GBK[33318] := 16#8C46;
   // UNICODE_TO_GBK[33319] := 16#B6B9;
   // UNICODE_TO_GBK[33320] := 16#8C47;
   // UNICODE_TO_GBK[33321] := 16#F4F8;
   // UNICODE_TO_GBK[33322] := 16#8C48;
   // UNICODE_TO_GBK[33323] := 16#D84D;
   // UNICODE_TO_GBK[33324] := 16#8C49;
   // UNICODE_TO_GBK[33325] := 16#F4F9;
   // UNICODE_TO_GBK[33326] := 16#8C4A;
   // UNICODE_TO_GBK[33327] := 16#D84E;
   // UNICODE_TO_GBK[33328] := 16#8C4B;
   // UNICODE_TO_GBK[33329] := 16#D84F;
   // UNICODE_TO_GBK[33330] := 16#8C4C;
   // UNICODE_TO_GBK[33331] := 16#CDE3;
   // UNICODE_TO_GBK[33332] := 16#8C4D;
   // UNICODE_TO_GBK[33333] := 16#D850;
   // UNICODE_TO_GBK[33334] := 16#8C4E;
   // UNICODE_TO_GBK[33335] := 16#D851;
   // UNICODE_TO_GBK[33336] := 16#8C4F;
   // UNICODE_TO_GBK[33337] := 16#D852;
   // UNICODE_TO_GBK[33338] := 16#8C50;
   // UNICODE_TO_GBK[33339] := 16#D853;
   // UNICODE_TO_GBK[33340] := 16#8C51;
   // UNICODE_TO_GBK[33341] := 16#D854;
   // UNICODE_TO_GBK[33342] := 16#8C52;
   // UNICODE_TO_GBK[33343] := 16#D855;
   // UNICODE_TO_GBK[33344] := 16#8C53;
   // UNICODE_TO_GBK[33345] := 16#D856;
   // UNICODE_TO_GBK[33346] := 16#8C54;
   // UNICODE_TO_GBK[33347] := 16#D857;
   // UNICODE_TO_GBK[33348] := 16#8C55;
   // UNICODE_TO_GBK[33349] := 16#F5B9;
   // UNICODE_TO_GBK[33350] := 16#8C56;
   // UNICODE_TO_GBK[33351] := 16#D858;
   // UNICODE_TO_GBK[33352] := 16#8C57;
   // UNICODE_TO_GBK[33353] := 16#D859;
   // UNICODE_TO_GBK[33354] := 16#8C58;
   // UNICODE_TO_GBK[33355] := 16#D85A;
   // UNICODE_TO_GBK[33356] := 16#8C59;
   // UNICODE_TO_GBK[33357] := 16#D85B;
   // UNICODE_TO_GBK[33358] := 16#8C5A;
   // UNICODE_TO_GBK[33359] := 16#EBE0;
   // UNICODE_TO_GBK[33360] := 16#8C5B;
   // UNICODE_TO_GBK[33361] := 16#D85C;
   // UNICODE_TO_GBK[33362] := 16#8C5C;
   // UNICODE_TO_GBK[33363] := 16#D85D;
   // UNICODE_TO_GBK[33364] := 16#8C5D;
   // UNICODE_TO_GBK[33365] := 16#D85E;
   // UNICODE_TO_GBK[33366] := 16#8C5E;
   // UNICODE_TO_GBK[33367] := 16#D85F;
   // UNICODE_TO_GBK[33368] := 16#8C5F;
   // UNICODE_TO_GBK[33369] := 16#D860;
   // UNICODE_TO_GBK[33370] := 16#8C60;
   // UNICODE_TO_GBK[33371] := 16#D861;
   // UNICODE_TO_GBK[33372] := 16#8C61;
   // UNICODE_TO_GBK[33373] := 16#CFF3;
   // UNICODE_TO_GBK[33374] := 16#8C62;
   // UNICODE_TO_GBK[33375] := 16#BBBF;
   // UNICODE_TO_GBK[33376] := 16#8C63;
   // UNICODE_TO_GBK[33377] := 16#D862;
   // UNICODE_TO_GBK[33378] := 16#8C64;
   // UNICODE_TO_GBK[33379] := 16#D863;
   // UNICODE_TO_GBK[33380] := 16#8C65;
   // UNICODE_TO_GBK[33381] := 16#D864;
   // UNICODE_TO_GBK[33382] := 16#8C66;
   // UNICODE_TO_GBK[33383] := 16#D865;
   // UNICODE_TO_GBK[33384] := 16#8C67;
   // UNICODE_TO_GBK[33385] := 16#D866;
   // UNICODE_TO_GBK[33386] := 16#8C68;
   // UNICODE_TO_GBK[33387] := 16#D867;
   // UNICODE_TO_GBK[33388] := 16#8C69;
   // UNICODE_TO_GBK[33389] := 16#D868;
   // UNICODE_TO_GBK[33390] := 16#8C6A;
   // UNICODE_TO_GBK[33391] := 16#BAC0;
   // UNICODE_TO_GBK[33392] := 16#8C6B;
   // UNICODE_TO_GBK[33393] := 16#D4A5;
   // UNICODE_TO_GBK[33394] := 16#8C6C;
   // UNICODE_TO_GBK[33395] := 16#D869;
   // UNICODE_TO_GBK[33396] := 16#8C6D;
   // UNICODE_TO_GBK[33397] := 16#D86A;
   // UNICODE_TO_GBK[33398] := 16#8C6E;
   // UNICODE_TO_GBK[33399] := 16#D86B;
   // UNICODE_TO_GBK[33400] := 16#8C6F;
   // UNICODE_TO_GBK[33401] := 16#D86C;
   // UNICODE_TO_GBK[33402] := 16#8C70;
   // UNICODE_TO_GBK[33403] := 16#D86D;
   // UNICODE_TO_GBK[33404] := 16#8C71;
   // UNICODE_TO_GBK[33405] := 16#D86E;
   // UNICODE_TO_GBK[33406] := 16#8C72;
   // UNICODE_TO_GBK[33407] := 16#D86F;
   // UNICODE_TO_GBK[33408] := 16#8C73;
   // UNICODE_TO_GBK[33409] := 16#E1D9;
   // UNICODE_TO_GBK[33410] := 16#8C74;
   // UNICODE_TO_GBK[33411] := 16#D870;
   // UNICODE_TO_GBK[33412] := 16#8C75;
   // UNICODE_TO_GBK[33413] := 16#D871;
   // UNICODE_TO_GBK[33414] := 16#8C76;
   // UNICODE_TO_GBK[33415] := 16#D872;
   // UNICODE_TO_GBK[33416] := 16#8C77;
   // UNICODE_TO_GBK[33417] := 16#D873;
   // UNICODE_TO_GBK[33418] := 16#8C78;
   // UNICODE_TO_GBK[33419] := 16#F5F4;
   // UNICODE_TO_GBK[33420] := 16#8C79;
   // UNICODE_TO_GBK[33421] := 16#B1AA;
   // UNICODE_TO_GBK[33422] := 16#8C7A;
   // UNICODE_TO_GBK[33423] := 16#B2F2;
   // UNICODE_TO_GBK[33424] := 16#8C7B;
   // UNICODE_TO_GBK[33425] := 16#D874;
   // UNICODE_TO_GBK[33426] := 16#8C7C;
   // UNICODE_TO_GBK[33427] := 16#D875;
   // UNICODE_TO_GBK[33428] := 16#8C7D;
   // UNICODE_TO_GBK[33429] := 16#D876;
   // UNICODE_TO_GBK[33430] := 16#8C7E;
   // UNICODE_TO_GBK[33431] := 16#D877;
   // UNICODE_TO_GBK[33432] := 16#8C7F;
   // UNICODE_TO_GBK[33433] := 16#D878;
   // UNICODE_TO_GBK[33434] := 16#8C80;
   // UNICODE_TO_GBK[33435] := 16#D879;
   // UNICODE_TO_GBK[33436] := 16#8C81;
   // UNICODE_TO_GBK[33437] := 16#D87A;
   // UNICODE_TO_GBK[33438] := 16#8C82;
   // UNICODE_TO_GBK[33439] := 16#F5F5;
   // UNICODE_TO_GBK[33440] := 16#8C83;
   // UNICODE_TO_GBK[33441] := 16#D87B;
   // UNICODE_TO_GBK[33442] := 16#8C84;
   // UNICODE_TO_GBK[33443] := 16#D87C;
   // UNICODE_TO_GBK[33444] := 16#8C85;
   // UNICODE_TO_GBK[33445] := 16#F5F7;
   // UNICODE_TO_GBK[33446] := 16#8C86;
   // UNICODE_TO_GBK[33447] := 16#D87D;
   // UNICODE_TO_GBK[33448] := 16#8C87;
   // UNICODE_TO_GBK[33449] := 16#D87E;
   // UNICODE_TO_GBK[33450] := 16#8C88;
   // UNICODE_TO_GBK[33451] := 16#D880;
   // UNICODE_TO_GBK[33452] := 16#8C89;
   // UNICODE_TO_GBK[33453] := 16#BAD1;
   // UNICODE_TO_GBK[33454] := 16#8C8A;
   // UNICODE_TO_GBK[33455] := 16#F5F6;
   // UNICODE_TO_GBK[33456] := 16#8C8B;
   // UNICODE_TO_GBK[33457] := 16#D881;
   // UNICODE_TO_GBK[33458] := 16#8C8C;
   // UNICODE_TO_GBK[33459] := 16#C3B2;
   // UNICODE_TO_GBK[33460] := 16#8C8D;
   // UNICODE_TO_GBK[33461] := 16#D882;
   // UNICODE_TO_GBK[33462] := 16#8C8E;
   // UNICODE_TO_GBK[33463] := 16#D883;
   // UNICODE_TO_GBK[33464] := 16#8C8F;
   // UNICODE_TO_GBK[33465] := 16#D884;
   // UNICODE_TO_GBK[33466] := 16#8C90;
   // UNICODE_TO_GBK[33467] := 16#D885;
   // UNICODE_TO_GBK[33468] := 16#8C91;
   // UNICODE_TO_GBK[33469] := 16#D886;
   // UNICODE_TO_GBK[33470] := 16#8C92;
   // UNICODE_TO_GBK[33471] := 16#D887;
   // UNICODE_TO_GBK[33472] := 16#8C93;
   // UNICODE_TO_GBK[33473] := 16#D888;
   // UNICODE_TO_GBK[33474] := 16#8C94;
   // UNICODE_TO_GBK[33475] := 16#F5F9;
   // UNICODE_TO_GBK[33476] := 16#8C95;
   // UNICODE_TO_GBK[33477] := 16#D889;
   // UNICODE_TO_GBK[33478] := 16#8C96;
   // UNICODE_TO_GBK[33479] := 16#D88A;
   // UNICODE_TO_GBK[33480] := 16#8C97;
   // UNICODE_TO_GBK[33481] := 16#D88B;
   // UNICODE_TO_GBK[33482] := 16#8C98;
   // UNICODE_TO_GBK[33483] := 16#F5F8;
   // UNICODE_TO_GBK[33484] := 16#8C99;
   // UNICODE_TO_GBK[33485] := 16#D88C;
   // UNICODE_TO_GBK[33486] := 16#8C9A;
   // UNICODE_TO_GBK[33487] := 16#D88D;
   // UNICODE_TO_GBK[33488] := 16#8C9B;
   // UNICODE_TO_GBK[33489] := 16#D88E;
   // UNICODE_TO_GBK[33490] := 16#8C9C;
   // UNICODE_TO_GBK[33491] := 16#D88F;
   // UNICODE_TO_GBK[33492] := 16#8C9D;
   // UNICODE_TO_GBK[33493] := 16#D890;
   // UNICODE_TO_GBK[33494] := 16#8C9E;
   // UNICODE_TO_GBK[33495] := 16#D891;
   // UNICODE_TO_GBK[33496] := 16#8C9F;
   // UNICODE_TO_GBK[33497] := 16#D892;
   // UNICODE_TO_GBK[33498] := 16#8CA0;
   // UNICODE_TO_GBK[33499] := 16#D893;
   // UNICODE_TO_GBK[33500] := 16#8CA1;
   // UNICODE_TO_GBK[33501] := 16#D894;
   // UNICODE_TO_GBK[33502] := 16#8CA2;
   // UNICODE_TO_GBK[33503] := 16#D895;
   // UNICODE_TO_GBK[33504] := 16#8CA3;
   // UNICODE_TO_GBK[33505] := 16#D896;
   // UNICODE_TO_GBK[33506] := 16#8CA4;
   // UNICODE_TO_GBK[33507] := 16#D897;
   // UNICODE_TO_GBK[33508] := 16#8CA5;
   // UNICODE_TO_GBK[33509] := 16#D898;
   // UNICODE_TO_GBK[33510] := 16#8CA6;
   // UNICODE_TO_GBK[33511] := 16#D899;
   // UNICODE_TO_GBK[33512] := 16#8CA7;
   // UNICODE_TO_GBK[33513] := 16#D89A;
   // UNICODE_TO_GBK[33514] := 16#8CA8;
   // UNICODE_TO_GBK[33515] := 16#D89B;
   // UNICODE_TO_GBK[33516] := 16#8CA9;
   // UNICODE_TO_GBK[33517] := 16#D89C;
   // UNICODE_TO_GBK[33518] := 16#8CAA;
   // UNICODE_TO_GBK[33519] := 16#D89D;
   // UNICODE_TO_GBK[33520] := 16#8CAB;
   // UNICODE_TO_GBK[33521] := 16#D89E;
   // UNICODE_TO_GBK[33522] := 16#8CAC;
   // UNICODE_TO_GBK[33523] := 16#D89F;
   // UNICODE_TO_GBK[33524] := 16#8CAD;
   // UNICODE_TO_GBK[33525] := 16#D8A0;
   // UNICODE_TO_GBK[33526] := 16#8CAE;
   // UNICODE_TO_GBK[33527] := 16#D940;
   // UNICODE_TO_GBK[33528] := 16#8CAF;
   // UNICODE_TO_GBK[33529] := 16#D941;
   // UNICODE_TO_GBK[33530] := 16#8CB0;
   // UNICODE_TO_GBK[33531] := 16#D942;
   // UNICODE_TO_GBK[33532] := 16#8CB1;
   // UNICODE_TO_GBK[33533] := 16#D943;
   // UNICODE_TO_GBK[33534] := 16#8CB2;
   // UNICODE_TO_GBK[33535] := 16#D944;
   // UNICODE_TO_GBK[33536] := 16#8CB3;
   // UNICODE_TO_GBK[33537] := 16#D945;
   // UNICODE_TO_GBK[33538] := 16#8CB4;
   // UNICODE_TO_GBK[33539] := 16#D946;
   // UNICODE_TO_GBK[33540] := 16#8CB5;
   // UNICODE_TO_GBK[33541] := 16#D947;
   // UNICODE_TO_GBK[33542] := 16#8CB6;
   // UNICODE_TO_GBK[33543] := 16#D948;
   // UNICODE_TO_GBK[33544] := 16#8CB7;
   // UNICODE_TO_GBK[33545] := 16#D949;
   // UNICODE_TO_GBK[33546] := 16#8CB8;
   // UNICODE_TO_GBK[33547] := 16#D94A;
   // UNICODE_TO_GBK[33548] := 16#8CB9;
   // UNICODE_TO_GBK[33549] := 16#D94B;
   // UNICODE_TO_GBK[33550] := 16#8CBA;
   // UNICODE_TO_GBK[33551] := 16#D94C;
   // UNICODE_TO_GBK[33552] := 16#8CBB;
   // UNICODE_TO_GBK[33553] := 16#D94D;
   // UNICODE_TO_GBK[33554] := 16#8CBC;
   // UNICODE_TO_GBK[33555] := 16#D94E;
   // UNICODE_TO_GBK[33556] := 16#8CBD;
   // UNICODE_TO_GBK[33557] := 16#D94F;
   // UNICODE_TO_GBK[33558] := 16#8CBE;
   // UNICODE_TO_GBK[33559] := 16#D950;
   // UNICODE_TO_GBK[33560] := 16#8CBF;
   // UNICODE_TO_GBK[33561] := 16#D951;
   // UNICODE_TO_GBK[33562] := 16#8CC0;
   // UNICODE_TO_GBK[33563] := 16#D952;
   // UNICODE_TO_GBK[33564] := 16#8CC1;
   // UNICODE_TO_GBK[33565] := 16#D953;
   // UNICODE_TO_GBK[33566] := 16#8CC2;
   // UNICODE_TO_GBK[33567] := 16#D954;
   // UNICODE_TO_GBK[33568] := 16#8CC3;
   // UNICODE_TO_GBK[33569] := 16#D955;
   // UNICODE_TO_GBK[33570] := 16#8CC4;
   // UNICODE_TO_GBK[33571] := 16#D956;
   // UNICODE_TO_GBK[33572] := 16#8CC5;
   // UNICODE_TO_GBK[33573] := 16#D957;
   // UNICODE_TO_GBK[33574] := 16#8CC6;
   // UNICODE_TO_GBK[33575] := 16#D958;
   // UNICODE_TO_GBK[33576] := 16#8CC7;
   // UNICODE_TO_GBK[33577] := 16#D959;
   // UNICODE_TO_GBK[33578] := 16#8CC8;
   // UNICODE_TO_GBK[33579] := 16#D95A;
   // UNICODE_TO_GBK[33580] := 16#8CC9;
   // UNICODE_TO_GBK[33581] := 16#D95B;
   // UNICODE_TO_GBK[33582] := 16#8CCA;
   // UNICODE_TO_GBK[33583] := 16#D95C;
   // UNICODE_TO_GBK[33584] := 16#8CCB;
   // UNICODE_TO_GBK[33585] := 16#D95D;
   // UNICODE_TO_GBK[33586] := 16#8CCC;
   // UNICODE_TO_GBK[33587] := 16#D95E;
   // UNICODE_TO_GBK[33588] := 16#8CCD;
   // UNICODE_TO_GBK[33589] := 16#D95F;
   // UNICODE_TO_GBK[33590] := 16#8CCE;
   // UNICODE_TO_GBK[33591] := 16#D960;
   // UNICODE_TO_GBK[33592] := 16#8CCF;
   // UNICODE_TO_GBK[33593] := 16#D961;
   // UNICODE_TO_GBK[33594] := 16#8CD0;
   // UNICODE_TO_GBK[33595] := 16#D962;
   // UNICODE_TO_GBK[33596] := 16#8CD1;
   // UNICODE_TO_GBK[33597] := 16#D963;
   // UNICODE_TO_GBK[33598] := 16#8CD2;
   // UNICODE_TO_GBK[33599] := 16#D964;
   // UNICODE_TO_GBK[33600] := 16#8CD3;
   // UNICODE_TO_GBK[33601] := 16#D965;
   // UNICODE_TO_GBK[33602] := 16#8CD4;
   // UNICODE_TO_GBK[33603] := 16#D966;
   // UNICODE_TO_GBK[33604] := 16#8CD5;
   // UNICODE_TO_GBK[33605] := 16#D967;
   // UNICODE_TO_GBK[33606] := 16#8CD6;
   // UNICODE_TO_GBK[33607] := 16#D968;
   // UNICODE_TO_GBK[33608] := 16#8CD7;
   // UNICODE_TO_GBK[33609] := 16#D969;
   // UNICODE_TO_GBK[33610] := 16#8CD8;
   // UNICODE_TO_GBK[33611] := 16#D96A;
   // UNICODE_TO_GBK[33612] := 16#8CD9;
   // UNICODE_TO_GBK[33613] := 16#D96B;
   // UNICODE_TO_GBK[33614] := 16#8CDA;
   // UNICODE_TO_GBK[33615] := 16#D96C;
   // UNICODE_TO_GBK[33616] := 16#8CDB;
   // UNICODE_TO_GBK[33617] := 16#D96D;
   // UNICODE_TO_GBK[33618] := 16#8CDC;
   // UNICODE_TO_GBK[33619] := 16#D96E;
   // UNICODE_TO_GBK[33620] := 16#8CDD;
   // UNICODE_TO_GBK[33621] := 16#D96F;
   // UNICODE_TO_GBK[33622] := 16#8CDE;
   // UNICODE_TO_GBK[33623] := 16#D970;
   // UNICODE_TO_GBK[33624] := 16#8CDF;
   // UNICODE_TO_GBK[33625] := 16#D971;
   // UNICODE_TO_GBK[33626] := 16#8CE0;
   // UNICODE_TO_GBK[33627] := 16#D972;
   // UNICODE_TO_GBK[33628] := 16#8CE1;
   // UNICODE_TO_GBK[33629] := 16#D973;
   // UNICODE_TO_GBK[33630] := 16#8CE2;
   // UNICODE_TO_GBK[33631] := 16#D974;
   // UNICODE_TO_GBK[33632] := 16#8CE3;
   // UNICODE_TO_GBK[33633] := 16#D975;
   // UNICODE_TO_GBK[33634] := 16#8CE4;
   // UNICODE_TO_GBK[33635] := 16#D976;
   // UNICODE_TO_GBK[33636] := 16#8CE5;
   // UNICODE_TO_GBK[33637] := 16#D977;
   // UNICODE_TO_GBK[33638] := 16#8CE6;
   // UNICODE_TO_GBK[33639] := 16#D978;
   // UNICODE_TO_GBK[33640] := 16#8CE7;
   // UNICODE_TO_GBK[33641] := 16#D979;
   // UNICODE_TO_GBK[33642] := 16#8CE8;
   // UNICODE_TO_GBK[33643] := 16#D97A;
   // UNICODE_TO_GBK[33644] := 16#8CE9;
   // UNICODE_TO_GBK[33645] := 16#D97B;
   // UNICODE_TO_GBK[33646] := 16#8CEA;
   // UNICODE_TO_GBK[33647] := 16#D97C;
   // UNICODE_TO_GBK[33648] := 16#8CEB;
   // UNICODE_TO_GBK[33649] := 16#D97D;
   // UNICODE_TO_GBK[33650] := 16#8CEC;
   // UNICODE_TO_GBK[33651] := 16#D97E;
   // UNICODE_TO_GBK[33652] := 16#8CED;
   // UNICODE_TO_GBK[33653] := 16#D980;
   // UNICODE_TO_GBK[33654] := 16#8CEE;
   // UNICODE_TO_GBK[33655] := 16#D981;
   // UNICODE_TO_GBK[33656] := 16#8CEF;
   // UNICODE_TO_GBK[33657] := 16#D982;
   // UNICODE_TO_GBK[33658] := 16#8CF0;
   // UNICODE_TO_GBK[33659] := 16#D983;
   // UNICODE_TO_GBK[33660] := 16#8CF1;
   // UNICODE_TO_GBK[33661] := 16#D984;
   // UNICODE_TO_GBK[33662] := 16#8CF2;
   // UNICODE_TO_GBK[33663] := 16#D985;
   // UNICODE_TO_GBK[33664] := 16#8CF3;
   // UNICODE_TO_GBK[33665] := 16#D986;
   // UNICODE_TO_GBK[33666] := 16#8CF4;
   // UNICODE_TO_GBK[33667] := 16#D987;
   // UNICODE_TO_GBK[33668] := 16#8CF5;
   // UNICODE_TO_GBK[33669] := 16#D988;
   // UNICODE_TO_GBK[33670] := 16#8CF6;
   // UNICODE_TO_GBK[33671] := 16#D989;
   // UNICODE_TO_GBK[33672] := 16#8CF7;
   // UNICODE_TO_GBK[33673] := 16#D98A;
   // UNICODE_TO_GBK[33674] := 16#8CF8;
   // UNICODE_TO_GBK[33675] := 16#D98B;
   // UNICODE_TO_GBK[33676] := 16#8CF9;
   // UNICODE_TO_GBK[33677] := 16#D98C;
   // UNICODE_TO_GBK[33678] := 16#8CFA;
   // UNICODE_TO_GBK[33679] := 16#D98D;
   // UNICODE_TO_GBK[33680] := 16#8CFB;
   // UNICODE_TO_GBK[33681] := 16#D98E;
   // UNICODE_TO_GBK[33682] := 16#8CFC;
   // UNICODE_TO_GBK[33683] := 16#D98F;
   // UNICODE_TO_GBK[33684] := 16#8CFD;
   // UNICODE_TO_GBK[33685] := 16#D990;
   // UNICODE_TO_GBK[33686] := 16#8CFE;
   // UNICODE_TO_GBK[33687] := 16#D991;
   // UNICODE_TO_GBK[33688] := 16#8CFF;
   // UNICODE_TO_GBK[33689] := 16#D992;
   // UNICODE_TO_GBK[33690] := 16#8D00;
   // UNICODE_TO_GBK[33691] := 16#D993;
   // UNICODE_TO_GBK[33692] := 16#8D01;
   // UNICODE_TO_GBK[33693] := 16#D994;
   // UNICODE_TO_GBK[33694] := 16#8D02;
   // UNICODE_TO_GBK[33695] := 16#D995;
   // UNICODE_TO_GBK[33696] := 16#8D03;
   // UNICODE_TO_GBK[33697] := 16#D996;
   // UNICODE_TO_GBK[33698] := 16#8D04;
   // UNICODE_TO_GBK[33699] := 16#D997;
   // UNICODE_TO_GBK[33700] := 16#8D05;
   // UNICODE_TO_GBK[33701] := 16#D998;
   // UNICODE_TO_GBK[33702] := 16#8D06;
   // UNICODE_TO_GBK[33703] := 16#D999;
   // UNICODE_TO_GBK[33704] := 16#8D07;
   // UNICODE_TO_GBK[33705] := 16#D99A;
   // UNICODE_TO_GBK[33706] := 16#8D08;
   // UNICODE_TO_GBK[33707] := 16#D99B;
   // UNICODE_TO_GBK[33708] := 16#8D09;
   // UNICODE_TO_GBK[33709] := 16#D99C;
   // UNICODE_TO_GBK[33710] := 16#8D0A;
   // UNICODE_TO_GBK[33711] := 16#D99D;
   // UNICODE_TO_GBK[33712] := 16#8D0B;
   // UNICODE_TO_GBK[33713] := 16#D99E;
   // UNICODE_TO_GBK[33714] := 16#8D0C;
   // UNICODE_TO_GBK[33715] := 16#D99F;
   // UNICODE_TO_GBK[33716] := 16#8D0D;
   // UNICODE_TO_GBK[33717] := 16#D9A0;
   // UNICODE_TO_GBK[33718] := 16#8D0E;
   // UNICODE_TO_GBK[33719] := 16#DA40;
   // UNICODE_TO_GBK[33720] := 16#8D0F;
   // UNICODE_TO_GBK[33721] := 16#DA41;
   // UNICODE_TO_GBK[33722] := 16#8D10;
   // UNICODE_TO_GBK[33723] := 16#DA42;
   // UNICODE_TO_GBK[33724] := 16#8D11;
   // UNICODE_TO_GBK[33725] := 16#DA43;
   // UNICODE_TO_GBK[33726] := 16#8D12;
   // UNICODE_TO_GBK[33727] := 16#DA44;
   // UNICODE_TO_GBK[33728] := 16#8D13;
   // UNICODE_TO_GBK[33729] := 16#DA45;
   // UNICODE_TO_GBK[33730] := 16#8D14;
   // UNICODE_TO_GBK[33731] := 16#DA46;
   // UNICODE_TO_GBK[33732] := 16#8D15;
   // UNICODE_TO_GBK[33733] := 16#DA47;
   // UNICODE_TO_GBK[33734] := 16#8D16;
   // UNICODE_TO_GBK[33735] := 16#DA48;
   // UNICODE_TO_GBK[33736] := 16#8D17;
   // UNICODE_TO_GBK[33737] := 16#DA49;
   // UNICODE_TO_GBK[33738] := 16#8D18;
   // UNICODE_TO_GBK[33739] := 16#DA4A;
   // UNICODE_TO_GBK[33740] := 16#8D19;
   // UNICODE_TO_GBK[33741] := 16#DA4B;
   // UNICODE_TO_GBK[33742] := 16#8D1A;
   // UNICODE_TO_GBK[33743] := 16#DA4C;
   // UNICODE_TO_GBK[33744] := 16#8D1B;
   // UNICODE_TO_GBK[33745] := 16#DA4D;
   // UNICODE_TO_GBK[33746] := 16#8D1C;
   // UNICODE_TO_GBK[33747] := 16#DA4E;
   // UNICODE_TO_GBK[33748] := 16#8D1D;
   // UNICODE_TO_GBK[33749] := 16#B1B4;
   // UNICODE_TO_GBK[33750] := 16#8D1E;
   // UNICODE_TO_GBK[33751] := 16#D5EA;
   // UNICODE_TO_GBK[33752] := 16#8D1F;
   // UNICODE_TO_GBK[33753] := 16#B8BA;
   // UNICODE_TO_GBK[33754] := 16#8D20;
   // UNICODE_TO_GBK[33755] := 16#DA4F;
   // UNICODE_TO_GBK[33756] := 16#8D21;
   // UNICODE_TO_GBK[33757] := 16#B9B1;
   // UNICODE_TO_GBK[33758] := 16#8D22;
   // UNICODE_TO_GBK[33759] := 16#B2C6;
   // UNICODE_TO_GBK[33760] := 16#8D23;
   // UNICODE_TO_GBK[33761] := 16#D4F0;
   // UNICODE_TO_GBK[33762] := 16#8D24;
   // UNICODE_TO_GBK[33763] := 16#CFCD;
   // UNICODE_TO_GBK[33764] := 16#8D25;
   // UNICODE_TO_GBK[33765] := 16#B0DC;
   // UNICODE_TO_GBK[33766] := 16#8D26;
   // UNICODE_TO_GBK[33767] := 16#D5CB;
   // UNICODE_TO_GBK[33768] := 16#8D27;
   // UNICODE_TO_GBK[33769] := 16#BBF5;
   // UNICODE_TO_GBK[33770] := 16#8D28;
   // UNICODE_TO_GBK[33771] := 16#D6CA;
   // UNICODE_TO_GBK[33772] := 16#8D29;
   // UNICODE_TO_GBK[33773] := 16#B7B7;
   // UNICODE_TO_GBK[33774] := 16#8D2A;
   // UNICODE_TO_GBK[33775] := 16#CCB0;
   // UNICODE_TO_GBK[33776] := 16#8D2B;
   // UNICODE_TO_GBK[33777] := 16#C6B6;
   // UNICODE_TO_GBK[33778] := 16#8D2C;
   // UNICODE_TO_GBK[33779] := 16#B1E1;
   // UNICODE_TO_GBK[33780] := 16#8D2D;
   // UNICODE_TO_GBK[33781] := 16#B9BA;
   // UNICODE_TO_GBK[33782] := 16#8D2E;
   // UNICODE_TO_GBK[33783] := 16#D6FC;
   // UNICODE_TO_GBK[33784] := 16#8D2F;
   // UNICODE_TO_GBK[33785] := 16#B9E1;
   // UNICODE_TO_GBK[33786] := 16#8D30;
   // UNICODE_TO_GBK[33787] := 16#B7A1;
   // UNICODE_TO_GBK[33788] := 16#8D31;
   // UNICODE_TO_GBK[33789] := 16#BCFA;
   // UNICODE_TO_GBK[33790] := 16#8D32;
   // UNICODE_TO_GBK[33791] := 16#EADA;
   // UNICODE_TO_GBK[33792] := 16#8D33;
   // UNICODE_TO_GBK[33793] := 16#EADB;
   // UNICODE_TO_GBK[33794] := 16#8D34;
   // UNICODE_TO_GBK[33795] := 16#CCF9;
   // UNICODE_TO_GBK[33796] := 16#8D35;
   // UNICODE_TO_GBK[33797] := 16#B9F3;
   // UNICODE_TO_GBK[33798] := 16#8D36;
   // UNICODE_TO_GBK[33799] := 16#EADC;
   // UNICODE_TO_GBK[33800] := 16#8D37;
   // UNICODE_TO_GBK[33801] := 16#B4FB;
   // UNICODE_TO_GBK[33802] := 16#8D38;
   // UNICODE_TO_GBK[33803] := 16#C3B3;
   // UNICODE_TO_GBK[33804] := 16#8D39;
   // UNICODE_TO_GBK[33805] := 16#B7D1;
   // UNICODE_TO_GBK[33806] := 16#8D3A;
   // UNICODE_TO_GBK[33807] := 16#BAD8;
   // UNICODE_TO_GBK[33808] := 16#8D3B;
   // UNICODE_TO_GBK[33809] := 16#EADD;
   // UNICODE_TO_GBK[33810] := 16#8D3C;
   // UNICODE_TO_GBK[33811] := 16#D4F4;
   // UNICODE_TO_GBK[33812] := 16#8D3D;
   // UNICODE_TO_GBK[33813] := 16#EADE;
   // UNICODE_TO_GBK[33814] := 16#8D3E;
   // UNICODE_TO_GBK[33815] := 16#BCD6;
   // UNICODE_TO_GBK[33816] := 16#8D3F;
   // UNICODE_TO_GBK[33817] := 16#BBDF;
   // UNICODE_TO_GBK[33818] := 16#8D40;
   // UNICODE_TO_GBK[33819] := 16#EADF;
   // UNICODE_TO_GBK[33820] := 16#8D41;
   // UNICODE_TO_GBK[33821] := 16#C1DE;
   // UNICODE_TO_GBK[33822] := 16#8D42;
   // UNICODE_TO_GBK[33823] := 16#C2B8;
   // UNICODE_TO_GBK[33824] := 16#8D43;
   // UNICODE_TO_GBK[33825] := 16#D4DF;
   // UNICODE_TO_GBK[33826] := 16#8D44;
   // UNICODE_TO_GBK[33827] := 16#D7CA;
   // UNICODE_TO_GBK[33828] := 16#8D45;
   // UNICODE_TO_GBK[33829] := 16#EAE0;
   // UNICODE_TO_GBK[33830] := 16#8D46;
   // UNICODE_TO_GBK[33831] := 16#EAE1;
   // UNICODE_TO_GBK[33832] := 16#8D47;
   // UNICODE_TO_GBK[33833] := 16#EAE4;
   // UNICODE_TO_GBK[33834] := 16#8D48;
   // UNICODE_TO_GBK[33835] := 16#EAE2;
   // UNICODE_TO_GBK[33836] := 16#8D49;
   // UNICODE_TO_GBK[33837] := 16#EAE3;
   // UNICODE_TO_GBK[33838] := 16#8D4A;
   // UNICODE_TO_GBK[33839] := 16#C9DE;
   // UNICODE_TO_GBK[33840] := 16#8D4B;
   // UNICODE_TO_GBK[33841] := 16#B8B3;
   // UNICODE_TO_GBK[33842] := 16#8D4C;
   // UNICODE_TO_GBK[33843] := 16#B6C4;
   // UNICODE_TO_GBK[33844] := 16#8D4D;
   // UNICODE_TO_GBK[33845] := 16#EAE5;
   // UNICODE_TO_GBK[33846] := 16#8D4E;
   // UNICODE_TO_GBK[33847] := 16#CAEA;
   // UNICODE_TO_GBK[33848] := 16#8D4F;
   // UNICODE_TO_GBK[33849] := 16#C9CD;
   // UNICODE_TO_GBK[33850] := 16#8D50;
   // UNICODE_TO_GBK[33851] := 16#B4CD;
   // UNICODE_TO_GBK[33852] := 16#8D51;
   // UNICODE_TO_GBK[33853] := 16#DA50;
   // UNICODE_TO_GBK[33854] := 16#8D52;
   // UNICODE_TO_GBK[33855] := 16#DA51;
   // UNICODE_TO_GBK[33856] := 16#8D53;
   // UNICODE_TO_GBK[33857] := 16#E2D9;
   // UNICODE_TO_GBK[33858] := 16#8D54;
   // UNICODE_TO_GBK[33859] := 16#C5E2;
   // UNICODE_TO_GBK[33860] := 16#8D55;
   // UNICODE_TO_GBK[33861] := 16#EAE6;
   // UNICODE_TO_GBK[33862] := 16#8D56;
   // UNICODE_TO_GBK[33863] := 16#C0B5;
   // UNICODE_TO_GBK[33864] := 16#8D57;
   // UNICODE_TO_GBK[33865] := 16#DA52;
   // UNICODE_TO_GBK[33866] := 16#8D58;
   // UNICODE_TO_GBK[33867] := 16#D7B8;
   // UNICODE_TO_GBK[33868] := 16#8D59;
   // UNICODE_TO_GBK[33869] := 16#EAE7;
   // UNICODE_TO_GBK[33870] := 16#8D5A;
   // UNICODE_TO_GBK[33871] := 16#D7AC;
   // UNICODE_TO_GBK[33872] := 16#8D5B;
   // UNICODE_TO_GBK[33873] := 16#C8FC;
   // UNICODE_TO_GBK[33874] := 16#8D5C;
   // UNICODE_TO_GBK[33875] := 16#D8D3;
   // UNICODE_TO_GBK[33876] := 16#8D5D;
   // UNICODE_TO_GBK[33877] := 16#D8CD;
   // UNICODE_TO_GBK[33878] := 16#8D5E;
   // UNICODE_TO_GBK[33879] := 16#D4DE;
   // UNICODE_TO_GBK[33880] := 16#8D5F;
   // UNICODE_TO_GBK[33881] := 16#DA53;
   // UNICODE_TO_GBK[33882] := 16#8D60;
   // UNICODE_TO_GBK[33883] := 16#D4F9;
   // UNICODE_TO_GBK[33884] := 16#8D61;
   // UNICODE_TO_GBK[33885] := 16#C9C4;
   // UNICODE_TO_GBK[33886] := 16#8D62;
   // UNICODE_TO_GBK[33887] := 16#D3AE;
   // UNICODE_TO_GBK[33888] := 16#8D63;
   // UNICODE_TO_GBK[33889] := 16#B8D3;
   // UNICODE_TO_GBK[33890] := 16#8D64;
   // UNICODE_TO_GBK[33891] := 16#B3E0;
   // UNICODE_TO_GBK[33892] := 16#8D65;
   // UNICODE_TO_GBK[33893] := 16#DA54;
   // UNICODE_TO_GBK[33894] := 16#8D66;
   // UNICODE_TO_GBK[33895] := 16#C9E2;
   // UNICODE_TO_GBK[33896] := 16#8D67;
   // UNICODE_TO_GBK[33897] := 16#F4F6;
   // UNICODE_TO_GBK[33898] := 16#8D68;
   // UNICODE_TO_GBK[33899] := 16#DA55;
   // UNICODE_TO_GBK[33900] := 16#8D69;
   // UNICODE_TO_GBK[33901] := 16#DA56;
   // UNICODE_TO_GBK[33902] := 16#8D6A;
   // UNICODE_TO_GBK[33903] := 16#DA57;
   // UNICODE_TO_GBK[33904] := 16#8D6B;
   // UNICODE_TO_GBK[33905] := 16#BAD5;
   // UNICODE_TO_GBK[33906] := 16#8D6C;
   // UNICODE_TO_GBK[33907] := 16#DA58;
   // UNICODE_TO_GBK[33908] := 16#8D6D;
   // UNICODE_TO_GBK[33909] := 16#F4F7;
   // UNICODE_TO_GBK[33910] := 16#8D6E;
   // UNICODE_TO_GBK[33911] := 16#DA59;
   // UNICODE_TO_GBK[33912] := 16#8D6F;
   // UNICODE_TO_GBK[33913] := 16#DA5A;
   // UNICODE_TO_GBK[33914] := 16#8D70;
   // UNICODE_TO_GBK[33915] := 16#D7DF;
   // UNICODE_TO_GBK[33916] := 16#8D71;
   // UNICODE_TO_GBK[33917] := 16#DA5B;
   // UNICODE_TO_GBK[33918] := 16#8D72;
   // UNICODE_TO_GBK[33919] := 16#DA5C;
   // UNICODE_TO_GBK[33920] := 16#8D73;
   // UNICODE_TO_GBK[33921] := 16#F4F1;
   // UNICODE_TO_GBK[33922] := 16#8D74;
   // UNICODE_TO_GBK[33923] := 16#B8B0;
   // UNICODE_TO_GBK[33924] := 16#8D75;
   // UNICODE_TO_GBK[33925] := 16#D5D4;
   // UNICODE_TO_GBK[33926] := 16#8D76;
   // UNICODE_TO_GBK[33927] := 16#B8CF;
   // UNICODE_TO_GBK[33928] := 16#8D77;
   // UNICODE_TO_GBK[33929] := 16#C6F0;
   // UNICODE_TO_GBK[33930] := 16#8D78;
   // UNICODE_TO_GBK[33931] := 16#DA5D;
   // UNICODE_TO_GBK[33932] := 16#8D79;
   // UNICODE_TO_GBK[33933] := 16#DA5E;
   // UNICODE_TO_GBK[33934] := 16#8D7A;
   // UNICODE_TO_GBK[33935] := 16#DA5F;
   // UNICODE_TO_GBK[33936] := 16#8D7B;
   // UNICODE_TO_GBK[33937] := 16#DA60;
   // UNICODE_TO_GBK[33938] := 16#8D7C;
   // UNICODE_TO_GBK[33939] := 16#DA61;
   // UNICODE_TO_GBK[33940] := 16#8D7D;
   // UNICODE_TO_GBK[33941] := 16#DA62;
   // UNICODE_TO_GBK[33942] := 16#8D7E;
   // UNICODE_TO_GBK[33943] := 16#DA63;
   // UNICODE_TO_GBK[33944] := 16#8D7F;
   // UNICODE_TO_GBK[33945] := 16#DA64;
   // UNICODE_TO_GBK[33946] := 16#8D80;
   // UNICODE_TO_GBK[33947] := 16#DA65;
   // UNICODE_TO_GBK[33948] := 16#8D81;
   // UNICODE_TO_GBK[33949] := 16#B3C3;
   // UNICODE_TO_GBK[33950] := 16#8D82;
   // UNICODE_TO_GBK[33951] := 16#DA66;
   // UNICODE_TO_GBK[33952] := 16#8D83;
   // UNICODE_TO_GBK[33953] := 16#DA67;
   // UNICODE_TO_GBK[33954] := 16#8D84;
   // UNICODE_TO_GBK[33955] := 16#F4F2;
   // UNICODE_TO_GBK[33956] := 16#8D85;
   // UNICODE_TO_GBK[33957] := 16#B3AC;
   // UNICODE_TO_GBK[33958] := 16#8D86;
   // UNICODE_TO_GBK[33959] := 16#DA68;
   // UNICODE_TO_GBK[33960] := 16#8D87;
   // UNICODE_TO_GBK[33961] := 16#DA69;
   // UNICODE_TO_GBK[33962] := 16#8D88;
   // UNICODE_TO_GBK[33963] := 16#DA6A;
   // UNICODE_TO_GBK[33964] := 16#8D89;
   // UNICODE_TO_GBK[33965] := 16#DA6B;
   // UNICODE_TO_GBK[33966] := 16#8D8A;
   // UNICODE_TO_GBK[33967] := 16#D4BD;
   // UNICODE_TO_GBK[33968] := 16#8D8B;
   // UNICODE_TO_GBK[33969] := 16#C7F7;
   // UNICODE_TO_GBK[33970] := 16#8D8C;
   // UNICODE_TO_GBK[33971] := 16#DA6C;
   // UNICODE_TO_GBK[33972] := 16#8D8D;
   // UNICODE_TO_GBK[33973] := 16#DA6D;
   // UNICODE_TO_GBK[33974] := 16#8D8E;
   // UNICODE_TO_GBK[33975] := 16#DA6E;
   // UNICODE_TO_GBK[33976] := 16#8D8F;
   // UNICODE_TO_GBK[33977] := 16#DA6F;
   // UNICODE_TO_GBK[33978] := 16#8D90;
   // UNICODE_TO_GBK[33979] := 16#DA70;
   // UNICODE_TO_GBK[33980] := 16#8D91;
   // UNICODE_TO_GBK[33981] := 16#F4F4;
   // UNICODE_TO_GBK[33982] := 16#8D92;
   // UNICODE_TO_GBK[33983] := 16#DA71;
   // UNICODE_TO_GBK[33984] := 16#8D93;
   // UNICODE_TO_GBK[33985] := 16#DA72;
   // UNICODE_TO_GBK[33986] := 16#8D94;
   // UNICODE_TO_GBK[33987] := 16#F4F3;
   // UNICODE_TO_GBK[33988] := 16#8D95;
   // UNICODE_TO_GBK[33989] := 16#DA73;
   // UNICODE_TO_GBK[33990] := 16#8D96;
   // UNICODE_TO_GBK[33991] := 16#DA74;
   // UNICODE_TO_GBK[33992] := 16#8D97;
   // UNICODE_TO_GBK[33993] := 16#DA75;
   // UNICODE_TO_GBK[33994] := 16#8D98;
   // UNICODE_TO_GBK[33995] := 16#DA76;
   // UNICODE_TO_GBK[33996] := 16#8D99;
   // UNICODE_TO_GBK[33997] := 16#DA77;
   // UNICODE_TO_GBK[33998] := 16#8D9A;
   // UNICODE_TO_GBK[33999] := 16#DA78;
   // UNICODE_TO_GBK[34000] := 16#8D9B;
   // UNICODE_TO_GBK[34001] := 16#DA79;
   // UNICODE_TO_GBK[34002] := 16#8D9C;
   // UNICODE_TO_GBK[34003] := 16#DA7A;
   // UNICODE_TO_GBK[34004] := 16#8D9D;
   // UNICODE_TO_GBK[34005] := 16#DA7B;
   // UNICODE_TO_GBK[34006] := 16#8D9E;
   // UNICODE_TO_GBK[34007] := 16#DA7C;
   // UNICODE_TO_GBK[34008] := 16#8D9F;
   // UNICODE_TO_GBK[34009] := 16#CCCB;
   // UNICODE_TO_GBK[34010] := 16#8DA0;
   // UNICODE_TO_GBK[34011] := 16#DA7D;
   // UNICODE_TO_GBK[34012] := 16#8DA1;
   // UNICODE_TO_GBK[34013] := 16#DA7E;
   // UNICODE_TO_GBK[34014] := 16#8DA2;
   // UNICODE_TO_GBK[34015] := 16#DA80;
   // UNICODE_TO_GBK[34016] := 16#8DA3;
   // UNICODE_TO_GBK[34017] := 16#C8A4;
   // UNICODE_TO_GBK[34018] := 16#8DA4;
   // UNICODE_TO_GBK[34019] := 16#DA81;
   // UNICODE_TO_GBK[34020] := 16#8DA5;
   // UNICODE_TO_GBK[34021] := 16#DA82;
   // UNICODE_TO_GBK[34022] := 16#8DA6;
   // UNICODE_TO_GBK[34023] := 16#DA83;
   // UNICODE_TO_GBK[34024] := 16#8DA7;
   // UNICODE_TO_GBK[34025] := 16#DA84;
   // UNICODE_TO_GBK[34026] := 16#8DA8;
   // UNICODE_TO_GBK[34027] := 16#DA85;
   // UNICODE_TO_GBK[34028] := 16#8DA9;
   // UNICODE_TO_GBK[34029] := 16#DA86;
   // UNICODE_TO_GBK[34030] := 16#8DAA;
   // UNICODE_TO_GBK[34031] := 16#DA87;
   // UNICODE_TO_GBK[34032] := 16#8DAB;
   // UNICODE_TO_GBK[34033] := 16#DA88;
   // UNICODE_TO_GBK[34034] := 16#8DAC;
   // UNICODE_TO_GBK[34035] := 16#DA89;
   // UNICODE_TO_GBK[34036] := 16#8DAD;
   // UNICODE_TO_GBK[34037] := 16#DA8A;
   // UNICODE_TO_GBK[34038] := 16#8DAE;
   // UNICODE_TO_GBK[34039] := 16#DA8B;
   // UNICODE_TO_GBK[34040] := 16#8DAF;
   // UNICODE_TO_GBK[34041] := 16#DA8C;
   // UNICODE_TO_GBK[34042] := 16#8DB0;
   // UNICODE_TO_GBK[34043] := 16#DA8D;
   // UNICODE_TO_GBK[34044] := 16#8DB1;
   // UNICODE_TO_GBK[34045] := 16#F4F5;
   // UNICODE_TO_GBK[34046] := 16#8DB2;
   // UNICODE_TO_GBK[34047] := 16#DA8E;
   // UNICODE_TO_GBK[34048] := 16#8DB3;
   // UNICODE_TO_GBK[34049] := 16#D7E3;
   // UNICODE_TO_GBK[34050] := 16#8DB4;
   // UNICODE_TO_GBK[34051] := 16#C5BF;
   // UNICODE_TO_GBK[34052] := 16#8DB5;
   // UNICODE_TO_GBK[34053] := 16#F5C0;
   // UNICODE_TO_GBK[34054] := 16#8DB6;
   // UNICODE_TO_GBK[34055] := 16#DA8F;
   // UNICODE_TO_GBK[34056] := 16#8DB7;
   // UNICODE_TO_GBK[34057] := 16#DA90;
   // UNICODE_TO_GBK[34058] := 16#8DB8;
   // UNICODE_TO_GBK[34059] := 16#F5BB;
   // UNICODE_TO_GBK[34060] := 16#8DB9;
   // UNICODE_TO_GBK[34061] := 16#DA91;
   // UNICODE_TO_GBK[34062] := 16#8DBA;
   // UNICODE_TO_GBK[34063] := 16#F5C3;
   // UNICODE_TO_GBK[34064] := 16#8DBB;
   // UNICODE_TO_GBK[34065] := 16#DA92;
   // UNICODE_TO_GBK[34066] := 16#8DBC;
   // UNICODE_TO_GBK[34067] := 16#F5C2;
   // UNICODE_TO_GBK[34068] := 16#8DBD;
   // UNICODE_TO_GBK[34069] := 16#DA93;
   // UNICODE_TO_GBK[34070] := 16#8DBE;
   // UNICODE_TO_GBK[34071] := 16#D6BA;
   // UNICODE_TO_GBK[34072] := 16#8DBF;
   // UNICODE_TO_GBK[34073] := 16#F5C1;
   // UNICODE_TO_GBK[34074] := 16#8DC0;
   // UNICODE_TO_GBK[34075] := 16#DA94;
   // UNICODE_TO_GBK[34076] := 16#8DC1;
   // UNICODE_TO_GBK[34077] := 16#DA95;
   // UNICODE_TO_GBK[34078] := 16#8DC2;
   // UNICODE_TO_GBK[34079] := 16#DA96;
   // UNICODE_TO_GBK[34080] := 16#8DC3;
   // UNICODE_TO_GBK[34081] := 16#D4BE;
   // UNICODE_TO_GBK[34082] := 16#8DC4;
   // UNICODE_TO_GBK[34083] := 16#F5C4;
   // UNICODE_TO_GBK[34084] := 16#8DC5;
   // UNICODE_TO_GBK[34085] := 16#DA97;
   // UNICODE_TO_GBK[34086] := 16#8DC6;
   // UNICODE_TO_GBK[34087] := 16#F5CC;
   // UNICODE_TO_GBK[34088] := 16#8DC7;
   // UNICODE_TO_GBK[34089] := 16#DA98;
   // UNICODE_TO_GBK[34090] := 16#8DC8;
   // UNICODE_TO_GBK[34091] := 16#DA99;
   // UNICODE_TO_GBK[34092] := 16#8DC9;
   // UNICODE_TO_GBK[34093] := 16#DA9A;
   // UNICODE_TO_GBK[34094] := 16#8DCA;
   // UNICODE_TO_GBK[34095] := 16#DA9B;
   // UNICODE_TO_GBK[34096] := 16#8DCB;
   // UNICODE_TO_GBK[34097] := 16#B0CF;
   // UNICODE_TO_GBK[34098] := 16#8DCC;
   // UNICODE_TO_GBK[34099] := 16#B5F8;
   // UNICODE_TO_GBK[34100] := 16#8DCD;
   // UNICODE_TO_GBK[34101] := 16#DA9C;
   // UNICODE_TO_GBK[34102] := 16#8DCE;
   // UNICODE_TO_GBK[34103] := 16#F5C9;
   // UNICODE_TO_GBK[34104] := 16#8DCF;
   // UNICODE_TO_GBK[34105] := 16#F5CA;
   // UNICODE_TO_GBK[34106] := 16#8DD0;
   // UNICODE_TO_GBK[34107] := 16#DA9D;
   // UNICODE_TO_GBK[34108] := 16#8DD1;
   // UNICODE_TO_GBK[34109] := 16#C5DC;
   // UNICODE_TO_GBK[34110] := 16#8DD2;
   // UNICODE_TO_GBK[34111] := 16#DA9E;
   // UNICODE_TO_GBK[34112] := 16#8DD3;
   // UNICODE_TO_GBK[34113] := 16#DA9F;
   // UNICODE_TO_GBK[34114] := 16#8DD4;
   // UNICODE_TO_GBK[34115] := 16#DAA0;
   // UNICODE_TO_GBK[34116] := 16#8DD5;
   // UNICODE_TO_GBK[34117] := 16#DB40;
   // UNICODE_TO_GBK[34118] := 16#8DD6;
   // UNICODE_TO_GBK[34119] := 16#F5C5;
   // UNICODE_TO_GBK[34120] := 16#8DD7;
   // UNICODE_TO_GBK[34121] := 16#F5C6;
   // UNICODE_TO_GBK[34122] := 16#8DD8;
   // UNICODE_TO_GBK[34123] := 16#DB41;
   // UNICODE_TO_GBK[34124] := 16#8DD9;
   // UNICODE_TO_GBK[34125] := 16#DB42;
   // UNICODE_TO_GBK[34126] := 16#8DDA;
   // UNICODE_TO_GBK[34127] := 16#F5C7;
   // UNICODE_TO_GBK[34128] := 16#8DDB;
   // UNICODE_TO_GBK[34129] := 16#F5CB;
   // UNICODE_TO_GBK[34130] := 16#8DDC;
   // UNICODE_TO_GBK[34131] := 16#DB43;
   // UNICODE_TO_GBK[34132] := 16#8DDD;
   // UNICODE_TO_GBK[34133] := 16#BEE0;
   // UNICODE_TO_GBK[34134] := 16#8DDE;
   // UNICODE_TO_GBK[34135] := 16#F5C8;
   // UNICODE_TO_GBK[34136] := 16#8DDF;
   // UNICODE_TO_GBK[34137] := 16#B8FA;
   // UNICODE_TO_GBK[34138] := 16#8DE0;
   // UNICODE_TO_GBK[34139] := 16#DB44;
   // UNICODE_TO_GBK[34140] := 16#8DE1;
   // UNICODE_TO_GBK[34141] := 16#DB45;
   // UNICODE_TO_GBK[34142] := 16#8DE2;
   // UNICODE_TO_GBK[34143] := 16#DB46;
   // UNICODE_TO_GBK[34144] := 16#8DE3;
   // UNICODE_TO_GBK[34145] := 16#F5D0;
   // UNICODE_TO_GBK[34146] := 16#8DE4;
   // UNICODE_TO_GBK[34147] := 16#F5D3;
   // UNICODE_TO_GBK[34148] := 16#8DE5;
   // UNICODE_TO_GBK[34149] := 16#DB47;
   // UNICODE_TO_GBK[34150] := 16#8DE6;
   // UNICODE_TO_GBK[34151] := 16#DB48;
   // UNICODE_TO_GBK[34152] := 16#8DE7;
   // UNICODE_TO_GBK[34153] := 16#DB49;
   // UNICODE_TO_GBK[34154] := 16#8DE8;
   // UNICODE_TO_GBK[34155] := 16#BFE7;
   // UNICODE_TO_GBK[34156] := 16#8DE9;
   // UNICODE_TO_GBK[34157] := 16#DB4A;
   // UNICODE_TO_GBK[34158] := 16#8DEA;
   // UNICODE_TO_GBK[34159] := 16#B9F2;
   // UNICODE_TO_GBK[34160] := 16#8DEB;
   // UNICODE_TO_GBK[34161] := 16#F5BC;
   // UNICODE_TO_GBK[34162] := 16#8DEC;
   // UNICODE_TO_GBK[34163] := 16#F5CD;
   // UNICODE_TO_GBK[34164] := 16#8DED;
   // UNICODE_TO_GBK[34165] := 16#DB4B;
   // UNICODE_TO_GBK[34166] := 16#8DEE;
   // UNICODE_TO_GBK[34167] := 16#DB4C;
   // UNICODE_TO_GBK[34168] := 16#8DEF;
   // UNICODE_TO_GBK[34169] := 16#C2B7;
   // UNICODE_TO_GBK[34170] := 16#8DF0;
   // UNICODE_TO_GBK[34171] := 16#DB4D;
   // UNICODE_TO_GBK[34172] := 16#8DF1;
   // UNICODE_TO_GBK[34173] := 16#DB4E;
   // UNICODE_TO_GBK[34174] := 16#8DF2;
   // UNICODE_TO_GBK[34175] := 16#DB4F;
   // UNICODE_TO_GBK[34176] := 16#8DF3;
   // UNICODE_TO_GBK[34177] := 16#CCF8;
   // UNICODE_TO_GBK[34178] := 16#8DF4;
   // UNICODE_TO_GBK[34179] := 16#DB50;
   // UNICODE_TO_GBK[34180] := 16#8DF5;
   // UNICODE_TO_GBK[34181] := 16#BCF9;
   // UNICODE_TO_GBK[34182] := 16#8DF6;
   // UNICODE_TO_GBK[34183] := 16#DB51;
   // UNICODE_TO_GBK[34184] := 16#8DF7;
   // UNICODE_TO_GBK[34185] := 16#F5CE;
   // UNICODE_TO_GBK[34186] := 16#8DF8;
   // UNICODE_TO_GBK[34187] := 16#F5CF;
   // UNICODE_TO_GBK[34188] := 16#8DF9;
   // UNICODE_TO_GBK[34189] := 16#F5D1;
   // UNICODE_TO_GBK[34190] := 16#8DFA;
   // UNICODE_TO_GBK[34191] := 16#B6E5;
   // UNICODE_TO_GBK[34192] := 16#8DFB;
   // UNICODE_TO_GBK[34193] := 16#F5D2;
   // UNICODE_TO_GBK[34194] := 16#8DFC;
   // UNICODE_TO_GBK[34195] := 16#DB52;
   // UNICODE_TO_GBK[34196] := 16#8DFD;
   // UNICODE_TO_GBK[34197] := 16#F5D5;
   // UNICODE_TO_GBK[34198] := 16#8DFE;
   // UNICODE_TO_GBK[34199] := 16#DB53;
   // UNICODE_TO_GBK[34200] := 16#8DFF;
   // UNICODE_TO_GBK[34201] := 16#DB54;
   // UNICODE_TO_GBK[34202] := 16#8E00;
   // UNICODE_TO_GBK[34203] := 16#DB55;
   // UNICODE_TO_GBK[34204] := 16#8E01;
   // UNICODE_TO_GBK[34205] := 16#DB56;
   // UNICODE_TO_GBK[34206] := 16#8E02;
   // UNICODE_TO_GBK[34207] := 16#DB57;
   // UNICODE_TO_GBK[34208] := 16#8E03;
   // UNICODE_TO_GBK[34209] := 16#DB58;
   // UNICODE_TO_GBK[34210] := 16#8E04;
   // UNICODE_TO_GBK[34211] := 16#DB59;
   // UNICODE_TO_GBK[34212] := 16#8E05;
   // UNICODE_TO_GBK[34213] := 16#F5BD;
   // UNICODE_TO_GBK[34214] := 16#8E06;
   // UNICODE_TO_GBK[34215] := 16#DB5A;
   // UNICODE_TO_GBK[34216] := 16#8E07;
   // UNICODE_TO_GBK[34217] := 16#DB5B;
   // UNICODE_TO_GBK[34218] := 16#8E08;
   // UNICODE_TO_GBK[34219] := 16#DB5C;
   // UNICODE_TO_GBK[34220] := 16#8E09;
   // UNICODE_TO_GBK[34221] := 16#F5D4;
   // UNICODE_TO_GBK[34222] := 16#8E0A;
   // UNICODE_TO_GBK[34223] := 16#D3BB;
   // UNICODE_TO_GBK[34224] := 16#8E0B;
   // UNICODE_TO_GBK[34225] := 16#DB5D;
   // UNICODE_TO_GBK[34226] := 16#8E0C;
   // UNICODE_TO_GBK[34227] := 16#B3EC;
   // UNICODE_TO_GBK[34228] := 16#8E0D;
   // UNICODE_TO_GBK[34229] := 16#DB5E;
   // UNICODE_TO_GBK[34230] := 16#8E0E;
   // UNICODE_TO_GBK[34231] := 16#DB5F;
   // UNICODE_TO_GBK[34232] := 16#8E0F;
   // UNICODE_TO_GBK[34233] := 16#CCA4;
   // UNICODE_TO_GBK[34234] := 16#8E10;
   // UNICODE_TO_GBK[34235] := 16#DB60;
   // UNICODE_TO_GBK[34236] := 16#8E11;
   // UNICODE_TO_GBK[34237] := 16#DB61;
   // UNICODE_TO_GBK[34238] := 16#8E12;
   // UNICODE_TO_GBK[34239] := 16#DB62;
   // UNICODE_TO_GBK[34240] := 16#8E13;
   // UNICODE_TO_GBK[34241] := 16#DB63;
   // UNICODE_TO_GBK[34242] := 16#8E14;
   // UNICODE_TO_GBK[34243] := 16#F5D6;
   // UNICODE_TO_GBK[34244] := 16#8E15;
   // UNICODE_TO_GBK[34245] := 16#DB64;
   // UNICODE_TO_GBK[34246] := 16#8E16;
   // UNICODE_TO_GBK[34247] := 16#DB65;
   // UNICODE_TO_GBK[34248] := 16#8E17;
   // UNICODE_TO_GBK[34249] := 16#DB66;
   // UNICODE_TO_GBK[34250] := 16#8E18;
   // UNICODE_TO_GBK[34251] := 16#DB67;
   // UNICODE_TO_GBK[34252] := 16#8E19;
   // UNICODE_TO_GBK[34253] := 16#DB68;
   // UNICODE_TO_GBK[34254] := 16#8E1A;
   // UNICODE_TO_GBK[34255] := 16#DB69;
   // UNICODE_TO_GBK[34256] := 16#8E1B;
   // UNICODE_TO_GBK[34257] := 16#DB6A;
   // UNICODE_TO_GBK[34258] := 16#8E1C;
   // UNICODE_TO_GBK[34259] := 16#DB6B;
   // UNICODE_TO_GBK[34260] := 16#8E1D;
   // UNICODE_TO_GBK[34261] := 16#F5D7;
   // UNICODE_TO_GBK[34262] := 16#8E1E;
   // UNICODE_TO_GBK[34263] := 16#BEE1;
   // UNICODE_TO_GBK[34264] := 16#8E1F;
   // UNICODE_TO_GBK[34265] := 16#F5D8;
   // UNICODE_TO_GBK[34266] := 16#8E20;
   // UNICODE_TO_GBK[34267] := 16#DB6C;
   // UNICODE_TO_GBK[34268] := 16#8E21;
   // UNICODE_TO_GBK[34269] := 16#DB6D;
   // UNICODE_TO_GBK[34270] := 16#8E22;
   // UNICODE_TO_GBK[34271] := 16#CCDF;
   // UNICODE_TO_GBK[34272] := 16#8E23;
   // UNICODE_TO_GBK[34273] := 16#F5DB;
   // UNICODE_TO_GBK[34274] := 16#8E24;
   // UNICODE_TO_GBK[34275] := 16#DB6E;
   // UNICODE_TO_GBK[34276] := 16#8E25;
   // UNICODE_TO_GBK[34277] := 16#DB6F;
   // UNICODE_TO_GBK[34278] := 16#8E26;
   // UNICODE_TO_GBK[34279] := 16#DB70;
   // UNICODE_TO_GBK[34280] := 16#8E27;
   // UNICODE_TO_GBK[34281] := 16#DB71;
   // UNICODE_TO_GBK[34282] := 16#8E28;
   // UNICODE_TO_GBK[34283] := 16#DB72;
   // UNICODE_TO_GBK[34284] := 16#8E29;
   // UNICODE_TO_GBK[34285] := 16#B2C8;
   // UNICODE_TO_GBK[34286] := 16#8E2A;
   // UNICODE_TO_GBK[34287] := 16#D7D9;
   // UNICODE_TO_GBK[34288] := 16#8E2B;
   // UNICODE_TO_GBK[34289] := 16#DB73;
   // UNICODE_TO_GBK[34290] := 16#8E2C;
   // UNICODE_TO_GBK[34291] := 16#F5D9;
   // UNICODE_TO_GBK[34292] := 16#8E2D;
   // UNICODE_TO_GBK[34293] := 16#DB74;
   // UNICODE_TO_GBK[34294] := 16#8E2E;
   // UNICODE_TO_GBK[34295] := 16#F5DA;
   // UNICODE_TO_GBK[34296] := 16#8E2F;
   // UNICODE_TO_GBK[34297] := 16#F5DC;
   // UNICODE_TO_GBK[34298] := 16#8E30;
   // UNICODE_TO_GBK[34299] := 16#DB75;
   // UNICODE_TO_GBK[34300] := 16#8E31;
   // UNICODE_TO_GBK[34301] := 16#F5E2;
   // UNICODE_TO_GBK[34302] := 16#8E32;
   // UNICODE_TO_GBK[34303] := 16#DB76;
   // UNICODE_TO_GBK[34304] := 16#8E33;
   // UNICODE_TO_GBK[34305] := 16#DB77;
   // UNICODE_TO_GBK[34306] := 16#8E34;
   // UNICODE_TO_GBK[34307] := 16#DB78;
   // UNICODE_TO_GBK[34308] := 16#8E35;
   // UNICODE_TO_GBK[34309] := 16#F5E0;
   // UNICODE_TO_GBK[34310] := 16#8E36;
   // UNICODE_TO_GBK[34311] := 16#DB79;
   // UNICODE_TO_GBK[34312] := 16#8E37;
   // UNICODE_TO_GBK[34313] := 16#DB7A;
   // UNICODE_TO_GBK[34314] := 16#8E38;
   // UNICODE_TO_GBK[34315] := 16#DB7B;
   // UNICODE_TO_GBK[34316] := 16#8E39;
   // UNICODE_TO_GBK[34317] := 16#F5DF;
   // UNICODE_TO_GBK[34318] := 16#8E3A;
   // UNICODE_TO_GBK[34319] := 16#F5DD;
   // UNICODE_TO_GBK[34320] := 16#8E3B;
   // UNICODE_TO_GBK[34321] := 16#DB7C;
   // UNICODE_TO_GBK[34322] := 16#8E3C;
   // UNICODE_TO_GBK[34323] := 16#DB7D;
   // UNICODE_TO_GBK[34324] := 16#8E3D;
   // UNICODE_TO_GBK[34325] := 16#F5E1;
   // UNICODE_TO_GBK[34326] := 16#8E3E;
   // UNICODE_TO_GBK[34327] := 16#DB7E;
   // UNICODE_TO_GBK[34328] := 16#8E3F;
   // UNICODE_TO_GBK[34329] := 16#DB80;
   // UNICODE_TO_GBK[34330] := 16#8E40;
   // UNICODE_TO_GBK[34331] := 16#F5DE;
   // UNICODE_TO_GBK[34332] := 16#8E41;
   // UNICODE_TO_GBK[34333] := 16#F5E4;
   // UNICODE_TO_GBK[34334] := 16#8E42;
   // UNICODE_TO_GBK[34335] := 16#F5E5;
   // UNICODE_TO_GBK[34336] := 16#8E43;
   // UNICODE_TO_GBK[34337] := 16#DB81;
   // UNICODE_TO_GBK[34338] := 16#8E44;
   // UNICODE_TO_GBK[34339] := 16#CCE3;
   // UNICODE_TO_GBK[34340] := 16#8E45;
   // UNICODE_TO_GBK[34341] := 16#DB82;
   // UNICODE_TO_GBK[34342] := 16#8E46;
   // UNICODE_TO_GBK[34343] := 16#DB83;
   // UNICODE_TO_GBK[34344] := 16#8E47;
   // UNICODE_TO_GBK[34345] := 16#E5BF;
   // UNICODE_TO_GBK[34346] := 16#8E48;
   // UNICODE_TO_GBK[34347] := 16#B5B8;
   // UNICODE_TO_GBK[34348] := 16#8E49;
   // UNICODE_TO_GBK[34349] := 16#F5E3;
   // UNICODE_TO_GBK[34350] := 16#8E4A;
   // UNICODE_TO_GBK[34351] := 16#F5E8;
   // UNICODE_TO_GBK[34352] := 16#8E4B;
   // UNICODE_TO_GBK[34353] := 16#CCA3;
   // UNICODE_TO_GBK[34354] := 16#8E4C;
   // UNICODE_TO_GBK[34355] := 16#DB84;
   // UNICODE_TO_GBK[34356] := 16#8E4D;
   // UNICODE_TO_GBK[34357] := 16#DB85;
   // UNICODE_TO_GBK[34358] := 16#8E4E;
   // UNICODE_TO_GBK[34359] := 16#DB86;
   // UNICODE_TO_GBK[34360] := 16#8E4F;
   // UNICODE_TO_GBK[34361] := 16#DB87;
   // UNICODE_TO_GBK[34362] := 16#8E50;
   // UNICODE_TO_GBK[34363] := 16#DB88;
   // UNICODE_TO_GBK[34364] := 16#8E51;
   // UNICODE_TO_GBK[34365] := 16#F5E6;
   // UNICODE_TO_GBK[34366] := 16#8E52;
   // UNICODE_TO_GBK[34367] := 16#F5E7;
   // UNICODE_TO_GBK[34368] := 16#8E53;
   // UNICODE_TO_GBK[34369] := 16#DB89;
   // UNICODE_TO_GBK[34370] := 16#8E54;
   // UNICODE_TO_GBK[34371] := 16#DB8A;
   // UNICODE_TO_GBK[34372] := 16#8E55;
   // UNICODE_TO_GBK[34373] := 16#DB8B;
   // UNICODE_TO_GBK[34374] := 16#8E56;
   // UNICODE_TO_GBK[34375] := 16#DB8C;
   // UNICODE_TO_GBK[34376] := 16#8E57;
   // UNICODE_TO_GBK[34377] := 16#DB8D;
   // UNICODE_TO_GBK[34378] := 16#8E58;
   // UNICODE_TO_GBK[34379] := 16#DB8E;
   // UNICODE_TO_GBK[34380] := 16#8E59;
   // UNICODE_TO_GBK[34381] := 16#F5BE;
   // UNICODE_TO_GBK[34382] := 16#8E5A;
   // UNICODE_TO_GBK[34383] := 16#DB8F;
   // UNICODE_TO_GBK[34384] := 16#8E5B;
   // UNICODE_TO_GBK[34385] := 16#DB90;
   // UNICODE_TO_GBK[34386] := 16#8E5C;
   // UNICODE_TO_GBK[34387] := 16#DB91;
   // UNICODE_TO_GBK[34388] := 16#8E5D;
   // UNICODE_TO_GBK[34389] := 16#DB92;
   // UNICODE_TO_GBK[34390] := 16#8E5E;
   // UNICODE_TO_GBK[34391] := 16#DB93;
   // UNICODE_TO_GBK[34392] := 16#8E5F;
   // UNICODE_TO_GBK[34393] := 16#DB94;
   // UNICODE_TO_GBK[34394] := 16#8E60;
   // UNICODE_TO_GBK[34395] := 16#DB95;
   // UNICODE_TO_GBK[34396] := 16#8E61;
   // UNICODE_TO_GBK[34397] := 16#DB96;
   // UNICODE_TO_GBK[34398] := 16#8E62;
   // UNICODE_TO_GBK[34399] := 16#DB97;
   // UNICODE_TO_GBK[34400] := 16#8E63;
   // UNICODE_TO_GBK[34401] := 16#DB98;
   // UNICODE_TO_GBK[34402] := 16#8E64;
   // UNICODE_TO_GBK[34403] := 16#DB99;
   // UNICODE_TO_GBK[34404] := 16#8E65;
   // UNICODE_TO_GBK[34405] := 16#DB9A;
   // UNICODE_TO_GBK[34406] := 16#8E66;
   // UNICODE_TO_GBK[34407] := 16#B1C4;
   // UNICODE_TO_GBK[34408] := 16#8E67;
   // UNICODE_TO_GBK[34409] := 16#DB9B;
   // UNICODE_TO_GBK[34410] := 16#8E68;
   // UNICODE_TO_GBK[34411] := 16#DB9C;
   // UNICODE_TO_GBK[34412] := 16#8E69;
   // UNICODE_TO_GBK[34413] := 16#F5BF;
   // UNICODE_TO_GBK[34414] := 16#8E6A;
   // UNICODE_TO_GBK[34415] := 16#DB9D;
   // UNICODE_TO_GBK[34416] := 16#8E6B;
   // UNICODE_TO_GBK[34417] := 16#DB9E;
   // UNICODE_TO_GBK[34418] := 16#8E6C;
   // UNICODE_TO_GBK[34419] := 16#B5C5;
   // UNICODE_TO_GBK[34420] := 16#8E6D;
   // UNICODE_TO_GBK[34421] := 16#B2E4;
   // UNICODE_TO_GBK[34422] := 16#8E6E;
   // UNICODE_TO_GBK[34423] := 16#DB9F;
   // UNICODE_TO_GBK[34424] := 16#8E6F;
   // UNICODE_TO_GBK[34425] := 16#F5EC;
   // UNICODE_TO_GBK[34426] := 16#8E70;
   // UNICODE_TO_GBK[34427] := 16#F5E9;
   // UNICODE_TO_GBK[34428] := 16#8E71;
   // UNICODE_TO_GBK[34429] := 16#DBA0;
   // UNICODE_TO_GBK[34430] := 16#8E72;
   // UNICODE_TO_GBK[34431] := 16#B6D7;
   // UNICODE_TO_GBK[34432] := 16#8E73;
   // UNICODE_TO_GBK[34433] := 16#DC40;
   // UNICODE_TO_GBK[34434] := 16#8E74;
   // UNICODE_TO_GBK[34435] := 16#F5ED;
   // UNICODE_TO_GBK[34436] := 16#8E75;
   // UNICODE_TO_GBK[34437] := 16#DC41;
   // UNICODE_TO_GBK[34438] := 16#8E76;
   // UNICODE_TO_GBK[34439] := 16#F5EA;
   // UNICODE_TO_GBK[34440] := 16#8E77;
   // UNICODE_TO_GBK[34441] := 16#DC42;
   // UNICODE_TO_GBK[34442] := 16#8E78;
   // UNICODE_TO_GBK[34443] := 16#DC43;
   // UNICODE_TO_GBK[34444] := 16#8E79;
   // UNICODE_TO_GBK[34445] := 16#DC44;
   // UNICODE_TO_GBK[34446] := 16#8E7A;
   // UNICODE_TO_GBK[34447] := 16#DC45;
   // UNICODE_TO_GBK[34448] := 16#8E7B;
   // UNICODE_TO_GBK[34449] := 16#DC46;
   // UNICODE_TO_GBK[34450] := 16#8E7C;
   // UNICODE_TO_GBK[34451] := 16#F5EB;
   // UNICODE_TO_GBK[34452] := 16#8E7D;
   // UNICODE_TO_GBK[34453] := 16#DC47;
   // UNICODE_TO_GBK[34454] := 16#8E7E;
   // UNICODE_TO_GBK[34455] := 16#DC48;
   // UNICODE_TO_GBK[34456] := 16#8E7F;
   // UNICODE_TO_GBK[34457] := 16#B4DA;
   // UNICODE_TO_GBK[34458] := 16#8E80;
   // UNICODE_TO_GBK[34459] := 16#DC49;
   // UNICODE_TO_GBK[34460] := 16#8E81;
   // UNICODE_TO_GBK[34461] := 16#D4EA;
   // UNICODE_TO_GBK[34462] := 16#8E82;
   // UNICODE_TO_GBK[34463] := 16#DC4A;
   // UNICODE_TO_GBK[34464] := 16#8E83;
   // UNICODE_TO_GBK[34465] := 16#DC4B;
   // UNICODE_TO_GBK[34466] := 16#8E84;
   // UNICODE_TO_GBK[34467] := 16#DC4C;
   // UNICODE_TO_GBK[34468] := 16#8E85;
   // UNICODE_TO_GBK[34469] := 16#F5EE;
   // UNICODE_TO_GBK[34470] := 16#8E86;
   // UNICODE_TO_GBK[34471] := 16#DC4D;
   // UNICODE_TO_GBK[34472] := 16#8E87;
   // UNICODE_TO_GBK[34473] := 16#B3F9;
   // UNICODE_TO_GBK[34474] := 16#8E88;
   // UNICODE_TO_GBK[34475] := 16#DC4E;
   // UNICODE_TO_GBK[34476] := 16#8E89;
   // UNICODE_TO_GBK[34477] := 16#DC4F;
   // UNICODE_TO_GBK[34478] := 16#8E8A;
   // UNICODE_TO_GBK[34479] := 16#DC50;
   // UNICODE_TO_GBK[34480] := 16#8E8B;
   // UNICODE_TO_GBK[34481] := 16#DC51;
   // UNICODE_TO_GBK[34482] := 16#8E8C;
   // UNICODE_TO_GBK[34483] := 16#DC52;
   // UNICODE_TO_GBK[34484] := 16#8E8D;
   // UNICODE_TO_GBK[34485] := 16#DC53;
   // UNICODE_TO_GBK[34486] := 16#8E8E;
   // UNICODE_TO_GBK[34487] := 16#DC54;
   // UNICODE_TO_GBK[34488] := 16#8E8F;
   // UNICODE_TO_GBK[34489] := 16#F5EF;
   // UNICODE_TO_GBK[34490] := 16#8E90;
   // UNICODE_TO_GBK[34491] := 16#F5F1;
   // UNICODE_TO_GBK[34492] := 16#8E91;
   // UNICODE_TO_GBK[34493] := 16#DC55;
   // UNICODE_TO_GBK[34494] := 16#8E92;
   // UNICODE_TO_GBK[34495] := 16#DC56;
   // UNICODE_TO_GBK[34496] := 16#8E93;
   // UNICODE_TO_GBK[34497] := 16#DC57;
   // UNICODE_TO_GBK[34498] := 16#8E94;
   // UNICODE_TO_GBK[34499] := 16#F5F0;
   // UNICODE_TO_GBK[34500] := 16#8E95;
   // UNICODE_TO_GBK[34501] := 16#DC58;
   // UNICODE_TO_GBK[34502] := 16#8E96;
   // UNICODE_TO_GBK[34503] := 16#DC59;
   // UNICODE_TO_GBK[34504] := 16#8E97;
   // UNICODE_TO_GBK[34505] := 16#DC5A;
   // UNICODE_TO_GBK[34506] := 16#8E98;
   // UNICODE_TO_GBK[34507] := 16#DC5B;
   // UNICODE_TO_GBK[34508] := 16#8E99;
   // UNICODE_TO_GBK[34509] := 16#DC5C;
   // UNICODE_TO_GBK[34510] := 16#8E9A;
   // UNICODE_TO_GBK[34511] := 16#DC5D;
   // UNICODE_TO_GBK[34512] := 16#8E9B;
   // UNICODE_TO_GBK[34513] := 16#DC5E;
   // UNICODE_TO_GBK[34514] := 16#8E9C;
   // UNICODE_TO_GBK[34515] := 16#F5F2;
   // UNICODE_TO_GBK[34516] := 16#8E9D;
   // UNICODE_TO_GBK[34517] := 16#DC5F;
   // UNICODE_TO_GBK[34518] := 16#8E9E;
   // UNICODE_TO_GBK[34519] := 16#F5F3;
   // UNICODE_TO_GBK[34520] := 16#8E9F;
   // UNICODE_TO_GBK[34521] := 16#DC60;
   // UNICODE_TO_GBK[34522] := 16#8EA0;
   // UNICODE_TO_GBK[34523] := 16#DC61;
   // UNICODE_TO_GBK[34524] := 16#8EA1;
   // UNICODE_TO_GBK[34525] := 16#DC62;
   // UNICODE_TO_GBK[34526] := 16#8EA2;
   // UNICODE_TO_GBK[34527] := 16#DC63;
   // UNICODE_TO_GBK[34528] := 16#8EA3;
   // UNICODE_TO_GBK[34529] := 16#DC64;
   // UNICODE_TO_GBK[34530] := 16#8EA4;
   // UNICODE_TO_GBK[34531] := 16#DC65;
   // UNICODE_TO_GBK[34532] := 16#8EA5;
   // UNICODE_TO_GBK[34533] := 16#DC66;
   // UNICODE_TO_GBK[34534] := 16#8EA6;
   // UNICODE_TO_GBK[34535] := 16#DC67;
   // UNICODE_TO_GBK[34536] := 16#8EA7;
   // UNICODE_TO_GBK[34537] := 16#DC68;
   // UNICODE_TO_GBK[34538] := 16#8EA8;
   // UNICODE_TO_GBK[34539] := 16#DC69;
   // UNICODE_TO_GBK[34540] := 16#8EA9;
   // UNICODE_TO_GBK[34541] := 16#DC6A;
   // UNICODE_TO_GBK[34542] := 16#8EAA;
   // UNICODE_TO_GBK[34543] := 16#DC6B;
   // UNICODE_TO_GBK[34544] := 16#8EAB;
   // UNICODE_TO_GBK[34545] := 16#C9ED;
   // UNICODE_TO_GBK[34546] := 16#8EAC;
   // UNICODE_TO_GBK[34547] := 16#B9AA;
   // UNICODE_TO_GBK[34548] := 16#8EAD;
   // UNICODE_TO_GBK[34549] := 16#DC6C;
   // UNICODE_TO_GBK[34550] := 16#8EAE;
   // UNICODE_TO_GBK[34551] := 16#DC6D;
   // UNICODE_TO_GBK[34552] := 16#8EAF;
   // UNICODE_TO_GBK[34553] := 16#C7FB;
   // UNICODE_TO_GBK[34554] := 16#8EB0;
   // UNICODE_TO_GBK[34555] := 16#DC6E;
   // UNICODE_TO_GBK[34556] := 16#8EB1;
   // UNICODE_TO_GBK[34557] := 16#DC6F;
   // UNICODE_TO_GBK[34558] := 16#8EB2;
   // UNICODE_TO_GBK[34559] := 16#B6E3;
   // UNICODE_TO_GBK[34560] := 16#8EB3;
   // UNICODE_TO_GBK[34561] := 16#DC70;
   // UNICODE_TO_GBK[34562] := 16#8EB4;
   // UNICODE_TO_GBK[34563] := 16#DC71;
   // UNICODE_TO_GBK[34564] := 16#8EB5;
   // UNICODE_TO_GBK[34565] := 16#DC72;
   // UNICODE_TO_GBK[34566] := 16#8EB6;
   // UNICODE_TO_GBK[34567] := 16#DC73;
   // UNICODE_TO_GBK[34568] := 16#8EB7;
   // UNICODE_TO_GBK[34569] := 16#DC74;
   // UNICODE_TO_GBK[34570] := 16#8EB8;
   // UNICODE_TO_GBK[34571] := 16#DC75;
   // UNICODE_TO_GBK[34572] := 16#8EB9;
   // UNICODE_TO_GBK[34573] := 16#DC76;
   // UNICODE_TO_GBK[34574] := 16#8EBA;
   // UNICODE_TO_GBK[34575] := 16#CCC9;
   // UNICODE_TO_GBK[34576] := 16#8EBB;
   // UNICODE_TO_GBK[34577] := 16#DC77;
   // UNICODE_TO_GBK[34578] := 16#8EBC;
   // UNICODE_TO_GBK[34579] := 16#DC78;
   // UNICODE_TO_GBK[34580] := 16#8EBD;
   // UNICODE_TO_GBK[34581] := 16#DC79;
   // UNICODE_TO_GBK[34582] := 16#8EBE;
   // UNICODE_TO_GBK[34583] := 16#DC7A;
   // UNICODE_TO_GBK[34584] := 16#8EBF;
   // UNICODE_TO_GBK[34585] := 16#DC7B;
   // UNICODE_TO_GBK[34586] := 16#8EC0;
   // UNICODE_TO_GBK[34587] := 16#DC7C;
   // UNICODE_TO_GBK[34588] := 16#8EC1;
   // UNICODE_TO_GBK[34589] := 16#DC7D;
   // UNICODE_TO_GBK[34590] := 16#8EC2;
   // UNICODE_TO_GBK[34591] := 16#DC7E;
   // UNICODE_TO_GBK[34592] := 16#8EC3;
   // UNICODE_TO_GBK[34593] := 16#DC80;
   // UNICODE_TO_GBK[34594] := 16#8EC4;
   // UNICODE_TO_GBK[34595] := 16#DC81;
   // UNICODE_TO_GBK[34596] := 16#8EC5;
   // UNICODE_TO_GBK[34597] := 16#DC82;
   // UNICODE_TO_GBK[34598] := 16#8EC6;
   // UNICODE_TO_GBK[34599] := 16#DC83;
   // UNICODE_TO_GBK[34600] := 16#8EC7;
   // UNICODE_TO_GBK[34601] := 16#DC84;
   // UNICODE_TO_GBK[34602] := 16#8EC8;
   // UNICODE_TO_GBK[34603] := 16#DC85;
   // UNICODE_TO_GBK[34604] := 16#8EC9;
   // UNICODE_TO_GBK[34605] := 16#DC86;
   // UNICODE_TO_GBK[34606] := 16#8ECA;
   // UNICODE_TO_GBK[34607] := 16#DC87;
   // UNICODE_TO_GBK[34608] := 16#8ECB;
   // UNICODE_TO_GBK[34609] := 16#DC88;
   // UNICODE_TO_GBK[34610] := 16#8ECC;
   // UNICODE_TO_GBK[34611] := 16#DC89;
   // UNICODE_TO_GBK[34612] := 16#8ECD;
   // UNICODE_TO_GBK[34613] := 16#DC8A;
   // UNICODE_TO_GBK[34614] := 16#8ECE;
   // UNICODE_TO_GBK[34615] := 16#EAA6;
   // UNICODE_TO_GBK[34616] := 16#8ECF;
   // UNICODE_TO_GBK[34617] := 16#DC8B;
   // UNICODE_TO_GBK[34618] := 16#8ED0;
   // UNICODE_TO_GBK[34619] := 16#DC8C;
   // UNICODE_TO_GBK[34620] := 16#8ED1;
   // UNICODE_TO_GBK[34621] := 16#DC8D;
   // UNICODE_TO_GBK[34622] := 16#8ED2;
   // UNICODE_TO_GBK[34623] := 16#DC8E;
   // UNICODE_TO_GBK[34624] := 16#8ED3;
   // UNICODE_TO_GBK[34625] := 16#DC8F;
   // UNICODE_TO_GBK[34626] := 16#8ED4;
   // UNICODE_TO_GBK[34627] := 16#DC90;
   // UNICODE_TO_GBK[34628] := 16#8ED5;
   // UNICODE_TO_GBK[34629] := 16#DC91;
   // UNICODE_TO_GBK[34630] := 16#8ED6;
   // UNICODE_TO_GBK[34631] := 16#DC92;
   // UNICODE_TO_GBK[34632] := 16#8ED7;
   // UNICODE_TO_GBK[34633] := 16#DC93;
   // UNICODE_TO_GBK[34634] := 16#8ED8;
   // UNICODE_TO_GBK[34635] := 16#DC94;
   // UNICODE_TO_GBK[34636] := 16#8ED9;
   // UNICODE_TO_GBK[34637] := 16#DC95;
   // UNICODE_TO_GBK[34638] := 16#8EDA;
   // UNICODE_TO_GBK[34639] := 16#DC96;
   // UNICODE_TO_GBK[34640] := 16#8EDB;
   // UNICODE_TO_GBK[34641] := 16#DC97;
   // UNICODE_TO_GBK[34642] := 16#8EDC;
   // UNICODE_TO_GBK[34643] := 16#DC98;
   // UNICODE_TO_GBK[34644] := 16#8EDD;
   // UNICODE_TO_GBK[34645] := 16#DC99;
   // UNICODE_TO_GBK[34646] := 16#8EDE;
   // UNICODE_TO_GBK[34647] := 16#DC9A;
   // UNICODE_TO_GBK[34648] := 16#8EDF;
   // UNICODE_TO_GBK[34649] := 16#DC9B;
   // UNICODE_TO_GBK[34650] := 16#8EE0;
   // UNICODE_TO_GBK[34651] := 16#DC9C;
   // UNICODE_TO_GBK[34652] := 16#8EE1;
   // UNICODE_TO_GBK[34653] := 16#DC9D;
   // UNICODE_TO_GBK[34654] := 16#8EE2;
   // UNICODE_TO_GBK[34655] := 16#DC9E;
   // UNICODE_TO_GBK[34656] := 16#8EE3;
   // UNICODE_TO_GBK[34657] := 16#DC9F;
   // UNICODE_TO_GBK[34658] := 16#8EE4;
   // UNICODE_TO_GBK[34659] := 16#DCA0;
   // UNICODE_TO_GBK[34660] := 16#8EE5;
   // UNICODE_TO_GBK[34661] := 16#DD40;
   // UNICODE_TO_GBK[34662] := 16#8EE6;
   // UNICODE_TO_GBK[34663] := 16#DD41;
   // UNICODE_TO_GBK[34664] := 16#8EE7;
   // UNICODE_TO_GBK[34665] := 16#DD42;
   // UNICODE_TO_GBK[34666] := 16#8EE8;
   // UNICODE_TO_GBK[34667] := 16#DD43;
   // UNICODE_TO_GBK[34668] := 16#8EE9;
   // UNICODE_TO_GBK[34669] := 16#DD44;
   // UNICODE_TO_GBK[34670] := 16#8EEA;
   // UNICODE_TO_GBK[34671] := 16#DD45;
   // UNICODE_TO_GBK[34672] := 16#8EEB;
   // UNICODE_TO_GBK[34673] := 16#DD46;
   // UNICODE_TO_GBK[34674] := 16#8EEC;
   // UNICODE_TO_GBK[34675] := 16#DD47;
   // UNICODE_TO_GBK[34676] := 16#8EED;
   // UNICODE_TO_GBK[34677] := 16#DD48;
   // UNICODE_TO_GBK[34678] := 16#8EEE;
   // UNICODE_TO_GBK[34679] := 16#DD49;
   // UNICODE_TO_GBK[34680] := 16#8EEF;
   // UNICODE_TO_GBK[34681] := 16#DD4A;
   // UNICODE_TO_GBK[34682] := 16#8EF0;
   // UNICODE_TO_GBK[34683] := 16#DD4B;
   // UNICODE_TO_GBK[34684] := 16#8EF1;
   // UNICODE_TO_GBK[34685] := 16#DD4C;
   // UNICODE_TO_GBK[34686] := 16#8EF2;
   // UNICODE_TO_GBK[34687] := 16#DD4D;
   // UNICODE_TO_GBK[34688] := 16#8EF3;
   // UNICODE_TO_GBK[34689] := 16#DD4E;
   // UNICODE_TO_GBK[34690] := 16#8EF4;
   // UNICODE_TO_GBK[34691] := 16#DD4F;
   // UNICODE_TO_GBK[34692] := 16#8EF5;
   // UNICODE_TO_GBK[34693] := 16#DD50;
   // UNICODE_TO_GBK[34694] := 16#8EF6;
   // UNICODE_TO_GBK[34695] := 16#DD51;
   // UNICODE_TO_GBK[34696] := 16#8EF7;
   // UNICODE_TO_GBK[34697] := 16#DD52;
   // UNICODE_TO_GBK[34698] := 16#8EF8;
   // UNICODE_TO_GBK[34699] := 16#DD53;
   // UNICODE_TO_GBK[34700] := 16#8EF9;
   // UNICODE_TO_GBK[34701] := 16#DD54;
   // UNICODE_TO_GBK[34702] := 16#8EFA;
   // UNICODE_TO_GBK[34703] := 16#DD55;
   // UNICODE_TO_GBK[34704] := 16#8EFB;
   // UNICODE_TO_GBK[34705] := 16#DD56;
   // UNICODE_TO_GBK[34706] := 16#8EFC;
   // UNICODE_TO_GBK[34707] := 16#DD57;
   // UNICODE_TO_GBK[34708] := 16#8EFD;
   // UNICODE_TO_GBK[34709] := 16#DD58;
   // UNICODE_TO_GBK[34710] := 16#8EFE;
   // UNICODE_TO_GBK[34711] := 16#DD59;
   // UNICODE_TO_GBK[34712] := 16#8EFF;
   // UNICODE_TO_GBK[34713] := 16#DD5A;
   // UNICODE_TO_GBK[34714] := 16#8F00;
   // UNICODE_TO_GBK[34715] := 16#DD5B;
   // UNICODE_TO_GBK[34716] := 16#8F01;
   // UNICODE_TO_GBK[34717] := 16#DD5C;
   // UNICODE_TO_GBK[34718] := 16#8F02;
   // UNICODE_TO_GBK[34719] := 16#DD5D;
   // UNICODE_TO_GBK[34720] := 16#8F03;
   // UNICODE_TO_GBK[34721] := 16#DD5E;
   // UNICODE_TO_GBK[34722] := 16#8F04;
   // UNICODE_TO_GBK[34723] := 16#DD5F;
   // UNICODE_TO_GBK[34724] := 16#8F05;
   // UNICODE_TO_GBK[34725] := 16#DD60;
   // UNICODE_TO_GBK[34726] := 16#8F06;
   // UNICODE_TO_GBK[34727] := 16#DD61;
   // UNICODE_TO_GBK[34728] := 16#8F07;
   // UNICODE_TO_GBK[34729] := 16#DD62;
   // UNICODE_TO_GBK[34730] := 16#8F08;
   // UNICODE_TO_GBK[34731] := 16#DD63;
   // UNICODE_TO_GBK[34732] := 16#8F09;
   // UNICODE_TO_GBK[34733] := 16#DD64;
   // UNICODE_TO_GBK[34734] := 16#8F0A;
   // UNICODE_TO_GBK[34735] := 16#DD65;
   // UNICODE_TO_GBK[34736] := 16#8F0B;
   // UNICODE_TO_GBK[34737] := 16#DD66;
   // UNICODE_TO_GBK[34738] := 16#8F0C;
   // UNICODE_TO_GBK[34739] := 16#DD67;
   // UNICODE_TO_GBK[34740] := 16#8F0D;
   // UNICODE_TO_GBK[34741] := 16#DD68;
   // UNICODE_TO_GBK[34742] := 16#8F0E;
   // UNICODE_TO_GBK[34743] := 16#DD69;
   // UNICODE_TO_GBK[34744] := 16#8F0F;
   // UNICODE_TO_GBK[34745] := 16#DD6A;
   // UNICODE_TO_GBK[34746] := 16#8F10;
   // UNICODE_TO_GBK[34747] := 16#DD6B;
   // UNICODE_TO_GBK[34748] := 16#8F11;
   // UNICODE_TO_GBK[34749] := 16#DD6C;
   // UNICODE_TO_GBK[34750] := 16#8F12;
   // UNICODE_TO_GBK[34751] := 16#DD6D;
   // UNICODE_TO_GBK[34752] := 16#8F13;
   // UNICODE_TO_GBK[34753] := 16#DD6E;
   // UNICODE_TO_GBK[34754] := 16#8F14;
   // UNICODE_TO_GBK[34755] := 16#DD6F;
   // UNICODE_TO_GBK[34756] := 16#8F15;
   // UNICODE_TO_GBK[34757] := 16#DD70;
   // UNICODE_TO_GBK[34758] := 16#8F16;
   // UNICODE_TO_GBK[34759] := 16#DD71;
   // UNICODE_TO_GBK[34760] := 16#8F17;
   // UNICODE_TO_GBK[34761] := 16#DD72;
   // UNICODE_TO_GBK[34762] := 16#8F18;
   // UNICODE_TO_GBK[34763] := 16#DD73;
   // UNICODE_TO_GBK[34764] := 16#8F19;
   // UNICODE_TO_GBK[34765] := 16#DD74;
   // UNICODE_TO_GBK[34766] := 16#8F1A;
   // UNICODE_TO_GBK[34767] := 16#DD75;
   // UNICODE_TO_GBK[34768] := 16#8F1B;
   // UNICODE_TO_GBK[34769] := 16#DD76;
   // UNICODE_TO_GBK[34770] := 16#8F1C;
   // UNICODE_TO_GBK[34771] := 16#DD77;
   // UNICODE_TO_GBK[34772] := 16#8F1D;
   // UNICODE_TO_GBK[34773] := 16#DD78;
   // UNICODE_TO_GBK[34774] := 16#8F1E;
   // UNICODE_TO_GBK[34775] := 16#DD79;
   // UNICODE_TO_GBK[34776] := 16#8F1F;
   // UNICODE_TO_GBK[34777] := 16#DD7A;
   // UNICODE_TO_GBK[34778] := 16#8F20;
   // UNICODE_TO_GBK[34779] := 16#DD7B;
   // UNICODE_TO_GBK[34780] := 16#8F21;
   // UNICODE_TO_GBK[34781] := 16#DD7C;
   // UNICODE_TO_GBK[34782] := 16#8F22;
   // UNICODE_TO_GBK[34783] := 16#DD7D;
   // UNICODE_TO_GBK[34784] := 16#8F23;
   // UNICODE_TO_GBK[34785] := 16#DD7E;
   // UNICODE_TO_GBK[34786] := 16#8F24;
   // UNICODE_TO_GBK[34787] := 16#DD80;
   // UNICODE_TO_GBK[34788] := 16#8F25;
   // UNICODE_TO_GBK[34789] := 16#DD81;
   // UNICODE_TO_GBK[34790] := 16#8F26;
   // UNICODE_TO_GBK[34791] := 16#DD82;
   // UNICODE_TO_GBK[34792] := 16#8F27;
   // UNICODE_TO_GBK[34793] := 16#DD83;
   // UNICODE_TO_GBK[34794] := 16#8F28;
   // UNICODE_TO_GBK[34795] := 16#DD84;
   // UNICODE_TO_GBK[34796] := 16#8F29;
   // UNICODE_TO_GBK[34797] := 16#DD85;
   // UNICODE_TO_GBK[34798] := 16#8F2A;
   // UNICODE_TO_GBK[34799] := 16#DD86;
   // UNICODE_TO_GBK[34800] := 16#8F2B;
   // UNICODE_TO_GBK[34801] := 16#DD87;
   // UNICODE_TO_GBK[34802] := 16#8F2C;
   // UNICODE_TO_GBK[34803] := 16#DD88;
   // UNICODE_TO_GBK[34804] := 16#8F2D;
   // UNICODE_TO_GBK[34805] := 16#DD89;
   // UNICODE_TO_GBK[34806] := 16#8F2E;
   // UNICODE_TO_GBK[34807] := 16#DD8A;
   // UNICODE_TO_GBK[34808] := 16#8F2F;
   // UNICODE_TO_GBK[34809] := 16#DD8B;
   // UNICODE_TO_GBK[34810] := 16#8F30;
   // UNICODE_TO_GBK[34811] := 16#DD8C;
   // UNICODE_TO_GBK[34812] := 16#8F31;
   // UNICODE_TO_GBK[34813] := 16#DD8D;
   // UNICODE_TO_GBK[34814] := 16#8F32;
   // UNICODE_TO_GBK[34815] := 16#DD8E;
   // UNICODE_TO_GBK[34816] := 16#8F33;
   // UNICODE_TO_GBK[34817] := 16#DD8F;
   // UNICODE_TO_GBK[34818] := 16#8F34;
   // UNICODE_TO_GBK[34819] := 16#DD90;
   // UNICODE_TO_GBK[34820] := 16#8F35;
   // UNICODE_TO_GBK[34821] := 16#DD91;
   // UNICODE_TO_GBK[34822] := 16#8F36;
   // UNICODE_TO_GBK[34823] := 16#DD92;
   // UNICODE_TO_GBK[34824] := 16#8F37;
   // UNICODE_TO_GBK[34825] := 16#DD93;
